LIN {X 0,Y 445.278,Z 563.704,A -85,B 0,C 180,E1 20681.751,E2 20681.751} C_VEL
LIN {X 0,Y 446.014,Z 547.85,A -85,B 0,C 180,E1 20680.554,E2 20680.554} C_VEL
LIN {X 0,Y 446.635,Z 530.926,A -85,B 0,C 180,E1 20679.559,E2 20679.559} C_VEL
LIN {X 0,Y 447.095,Z 513.78,A -85,B 0,C 180,E1 20678.817,E2 20678.817} C_VEL
LIN {X 0,Y 447.348,Z 495.46,A -85,B 0,C 180,E1 20678.284,E2 20678.284} C_VEL
LIN {X 0,Y 449.909,Z 332.781,A -85,B 0,C 180,E1 20675.326,E2 20675.326} C_VEL
LIN {X 0,Y 449.103,Z 327.513,A -85,B 0,C 180,E1 20675.165,E2 20675.165} C_VEL
LIN {X 0,Y 450.293,Z 289.121,A -85,B 0,C 180,E1 20671.484,E2 20671.484} C_VEL
LIN {X 0,Y 450.643,Z 279.918,A -85,B 0,C 180,E1 20670.582,E2 20670.582} C_VEL
LIN {X 0,Y 452.131,Z 281.25,A -85,B 0,C 180,E1 20670.354,E2 20670.354} C_VEL
LIN {X 0,Y 454.578,Z 280.888,A -85,B 0,C 180,E1 20670.046,E2 20670.046} C_VEL
LIN {X 0,Y 458.108,Z 278.184,A -85,B 0,C 180,E1 20669.668,E2 20669.668} C_VEL
LIN {X 0,Y 459.445,Z 277.014,A -85,B 0,C 180,E1 20669.531,E2 20669.531} C_VEL
LIN {X 0,Y 463.235,Z 276.31,A -85,B 0,C 180,E1 20669.089,E2 20669.089} C_VEL
LIN {X 0,Y 467.513,Z 273.586,A -85,B 0,C 180,E1 20668.652,E2 20668.652} C_VEL
LIN {X 0,Y 468.934,Z 272.801,A -85,B 0,C 180,E1 20668.507,E2 20668.507} C_VEL
LIN {X 0,Y 471.015,Z 272.513,A -85,B 0,C 180,E1 20668.278,E2 20668.278} C_VEL
LIN {X 0,Y 466.209,Z 421.313,A -85,B 0,C 180,E1 20665.555,E2 20665.555} C_VEL
LIN {X 0,Y 465.176,Z 428.993,A -85,B 0,C 180,E1 20665.49,E2 20665.49} C_VEL
LIN {X 0,Y 459.547,Z 449.472,A -85,B 0,C 180,E1 20665.582,E2 20665.582} C_VEL
LIN {X 0,Y 458.739,Z 456.06,A -85,B 0,C 180,E1 20665.515,E2 20665.515} C_VEL
LIN {X 0,Y 457.752,Z 483.582,A -85,B 0,C 180,E1 20664.917,E2 20664.917} C_VEL
LIN {X 0,Y 456.588,Z 504.2,A -85,B 0,C 180,E1 20664.247,E2 20664.247} C_VEL
LIN {X 0,Y 454.896,Z 524.708,A -85,B 0,C 180,E1 20663.348,E2 20663.348} C_VEL
LIN {X 0,Y 452.943,Z 544.086,A -85,B 0,C 180,E1 20662.268,E2 20662.268} C_VEL
LIN {X 0,Y 450.644,Z 563.469,A -85,B 0,C 180,E1 20660.94,E2 20660.94} C_VEL
LIN {X 0,Y 448.195,Z 581.756,A -85,B 0,C 180,E1 20659.43,E2 20659.43} C_VEL
LIN {X 0,Y 445.575,Z 599.353,A -85,B 0,C 180,E1 20657.685,E2 20657.685} C_VEL
LIN {X 0,Y 443.037,Z 615.611,A -85,B 0,C 180,E1 20655.784,E2 20655.784} C_VEL
LIN {X 0,Y 440.527,Z 631.382,A -85,B 0,C 180,E1 20653.611,E2 20653.611} C_VEL
LIN {X 0,Y 438.339,Z 645.243,A -85,B 0,C 180,E1 20651.369,E2 20651.369} C_VEL
LIN {X 0,Y 436.373,Z 658.158,A -85,B 0,C 180,E1 20648.89,E2 20648.89} C_VEL
LIN {X 0,Y 434.733,Z 670.08,A -85,B 0,C 180,E1 20646.168,E2 20646.168} C_VEL
LIN {X 0,Y 433.546,Z 679.999,A -85,B 0,C 180,E1 20643.449,E2 20643.449} C_VEL
LIN {X 0,Y 432.699,Z 688.525,A -85,B 0,C 180,E1 20640.555,E2 20640.555} C_VEL
LIN {X 0,Y 432.258,Z 694.523,A -85,B 0,C 180,E1 20638.006,E2 20638.006} C_VEL
LIN {X 0,Y 432.009,Z 700.325,A -85,B 0,C 180,E1 20634.869,E2 20634.869} C_VEL
LIN {X 0,Y 431.939,Z 703.61,A -85,B 0,C 180,E1 20632.311,E2 20632.311} C_VEL
LIN {X 0,Y 431.908,Z 705.568,A -85,B 0,C 180,E1 20629.896,E2 20629.896} C_VEL
LIN {X 0,Y 431.906,Z 706.457,A -85,B 0,C 180,E1 20627.237,E2 20627.237} C_VEL
LIN {X 0,Y 431.914,Z 705.763,A -85,B 0,C 180,E1 20624.342,E2 20624.342} C_VEL
LIN {X 0,Y 431.928,Z 703.903,A -85,B 0,C 180,E1 20621.89,E2 20621.89} C_VEL
LIN {X 0,Y 431.98,Z 700.918,A -85,B 0,C 180,E1 20619.459,E2 20619.459} C_VEL
LIN {X 0,Y 432.211,Z 695.519,A -85,B 0,C 180,E1 20616.376,E2 20616.376} C_VEL
LIN {X 0,Y 432.599,Z 689.749,A -85,B 0,C 180,E1 20613.843,E2 20613.843} C_VEL
LIN {X 0,Y 433.329,Z 681.908,A -85,B 0,C 180,E1 20611.058,E2 20611.058} C_VEL
LIN {X 0,Y 434.437,Z 672.167,A -85,B 0,C 180,E1 20608.286,E2 20608.286} C_VEL
LIN {X 0,Y 435.841,Z 661.693,A -85,B 0,C 180,E1 20605.79,E2 20605.79} C_VEL
LIN {X 0,Y 437.776,Z 648.664,A -85,B 0,C 180,E1 20603.179,E2 20603.179} C_VEL
LIN {X 0,Y 440.074,Z 634.053,A -85,B 0,C 180,E1 20600.717,E2 20600.717} C_VEL
LIN {X 0,Y 442.535,Z 618.775,A -85,B 0,C 180,E1 20598.532,E2 20598.532} C_VEL
LIN {X 0,Y 445.057,Z 602.818,A -85,B 0,C 180,E1 20596.601,E2 20596.601} C_VEL
LIN {X 0,Y 447.614,Z 585.784,A -85,B 0,C 180,E1 20594.85,E2 20594.85} C_VEL
LIN {X 0,Y 450.175,Z 567.801,A -85,B 0,C 180,E1 20593.284,E2 20593.284} C_VEL
LIN {X 0,Y 452.464,Z 549.874,A -85,B 0,C 180,E1 20591.979,E2 20591.979} C_VEL
LIN {X 0,Y 454.464,Z 531.263,A -85,B 0,C 180,E1 20590.864,E2 20590.864} C_VEL
LIN {X 0,Y 456.333,Z 510.862,A -85,B 0,C 180,E1 20589.879,E2 20589.879} C_VEL
LIN {X 0,Y 457.832,Z 489.947,A -85,B 0,C 180,E1 20589.109,E2 20589.109} C_VEL
LIN {X 0,Y 458.748,Z 469.432,A -85,B 0,C 180,E1 20588.58,E2 20588.58} C_VEL
LIN {X 0,Y 465.748,Z 266.596,A -85,B 0,C 180,E1 20584.795,E2 20584.795} C_VEL
LIN {X 0,Y 466.581,Z 237.059,A -85,B 0,C 180,E1 20584.241,E2 20584.241} C_VEL
LIN {X 0,Y 453.17,Z 217.007,A -85,B 0,C 180,E1 20582.222,E2 20582.222} C_VEL
LIN {X 0,Y 445.587,Z 207.661,A -85,B 0,C 180,E1 20581.061,E2 20581.061} C_VEL
LIN {X 0,Y 440.176,Z 201.25,A -85,B 0,C 180,E1 20580.168,E2 20580.168} C_VEL
LIN {X 0,Y 437.829,Z 196.904,A -85,B 0,C 180,E1 20579.168,E2 20579.168} C_VEL
LIN {X 0,Y 435.976,Z 193.053,A -85,B 0,C 180,E1 20578.305,E2 20578.305} C_VEL
LIN {X 0,Y 433.608,Z 189.423,A -85,B 0,C 180,E1 20577.345,E2 20577.345} C_VEL
LIN {X 0,Y 433.237,Z 187.766,A -85,B 0,C 180,E1 20576.999,E2 20576.999} C_VEL
LIN {X 0,Y 433.227,Z 187.768,A -85,B 0,C 180,E1 20573.126,E2 20573.126} C_VEL
LIN {X 0,Y 433.243,Z 187.762,A -85,B 0,C 180,E1 20569.397,E2 20569.397} C_VEL
LIN {X 0,Y 433.252,Z 187.758,A -85,B 0,C 180,E1 20565.632,E2 20565.632} C_VEL
LIN {X 0,Y 433.251,Z 187.759,A -85,B 0,C 180,E1 20561.805,E2 20561.805} C_VEL
LIN {X 0,Y 433.236,Z 187.766,A -85,B 0,C 180,E1 20558.04,E2 20558.04} C_VEL
LIN {X 0,Y 433.219,Z 187.773,A -85,B 0,C 180,E1 20554.274,E2 20554.274} C_VEL
LIN {X 0,Y 433.244,Z 187.764,A -85,B 0,C 180,E1 20550.513,E2 20550.513} C_VEL
LIN {X 0,Y 433.259,Z 187.752,A -85,B 0,C 180,E1 20546.734,E2 20546.734} C_VEL
LIN {X 0,Y 433.251,Z 187.746,A -85,B 0,C 180,E1 20542.955,E2 20542.955} C_VEL
LIN {X 0,Y 433.235,Z 187.76,A -85,B 0,C 180,E1 20539.131,E2 20539.131} C_VEL
LIN {X 0,Y 433.207,Z 187.773,A -85,B 0,C 180,E1 20535.393,E2 20535.393} C_VEL
LIN {X 0,Y 433.2,Z 187.772,A -85,B 0,C 180,E1 20531.584,E2 20531.584} C_VEL
LIN {X 0,Y 433.222,Z 187.759,A -85,B 0,C 180,E1 20527.827,E2 20527.827} C_VEL
LIN {X 0,Y 433.245,Z 187.748,A -85,B 0,C 180,E1 20524.103,E2 20524.103} C_VEL
LIN {X 0,Y 433.258,Z 187.751,A -85,B 0,C 180,E1 20520.265,E2 20520.265} C_VEL
LIN {X 0,Y 433.251,Z 187.755,A -85,B 0,C 180,E1 20516.428,E2 20516.428} C_VEL
LIN {X 0,Y 433.235,Z 187.757,A -85,B 0,C 180,E1 20512.575,E2 20512.575} C_VEL
LIN {X 0,Y 433.248,Z 187.755,A -85,B 0,C 180,E1 20508.761,E2 20508.761} C_VEL
LIN {X 0,Y 433.262,Z 187.753,A -85,B 0,C 180,E1 20505.021,E2 20505.021} C_VEL
LIN {X 0,Y 433.248,Z 187.756,A -85,B 0,C 180,E1 20501.15,E2 20501.15} C_VEL
LIN {X 0,Y 433.488,Z 188.953,A -85,B 0,C 180,E1 20500.882,E2 20500.882} C_VEL
LIN {X 0,Y 435.26,Z 192.141,A -85,B 0,C 180,E1 20500.125,E2 20500.125} C_VEL
LIN {X 0,Y 436.158,Z 193.757,A -85,B 0,C 180,E1 20499.748,E2 20499.748} C_VEL
LIN {X 0,Y 438.842,Z 198.769,A -85,B 0,C 180,E1 20498.621,E2 20498.621} C_VEL
LIN {X 0,Y 443.751,Z 208.113,A -85,B 0,C 180,E1 20496.637,E2 20496.637} C_VEL
LIN {X 0,Y 450.114,Z 220.548,A -85,B 0,C 180,E1 20494.191,E2 20494.191} C_VEL
LIN {X 0,Y 458.928,Z 239.006,A -85,B 0,C 180,E1 20490.932,E2 20490.932} C_VEL
LIN {X 0,Y 465.596,Z 254.171,A -85,B 0,C 180,E1 20488.522,E2 20488.522} C_VEL
LIN {X 0,Y 461.582,Z 295.714,A -85,B 0,C 180,E1 20484.966,E2 20484.966} C_VEL
LIN {X 0,Y 460.595,Z 316.537,A -85,B 0,C 180,E1 20483.114,E2 20483.114} C_VEL
LIN {X 0,Y 461.621,Z 333.917,A -85,B 0,C 180,E1 20481.406,E2 20481.406} C_VEL
LIN {X 0,Y 464.524,Z 349.654,A -85,B 0,C 180,E1 20479.699,E2 20479.699} C_VEL
LIN {X 0,Y 469.216,Z 363.952,A -85,B 0,C 180,E1 20478.002,E2 20478.002} C_VEL
LIN {X 0,Y 475.939,Z 377.183,A -85,B 0,C 180,E1 20476.276,E2 20476.276} C_VEL
LIN {X 0,Y 484.496,Z 388.72,A -85,B 0,C 180,E1 20474.604,E2 20474.604} C_VEL
LIN {X 0,Y 493.529,Z 397.655,A -85,B 0,C 180,E1 20473.17,E2 20473.17} C_VEL
LIN {X 0,Y 501.232,Z 403.797,A -85,B 0,C 180,E1 20472.107,E2 20472.107} C_VEL
LIN {X 0,Y 490.067,Z 420.572,A -85,B 0,C 180,E1 20471.613,E2 20471.613} C_VEL
LIN {X 0,Y 481.918,Z 435.231,A -85,B 0,C 180,E1 20471.045,E2 20471.045} C_VEL
LIN {X 0,Y 472.016,Z 452.159,A -85,B 0,C 180,E1 20470.405,E2 20470.405} C_VEL
LIN {X 0,Y 465.347,Z 466.548,A -85,B 0,C 180,E1 20469.718,E2 20469.718} C_VEL
LIN {X 0,Y 463.803,Z 470.28,A -85,B 0,C 180,E1 20469.564,E2 20469.564} C_VEL
LIN {X 0,Y 461.689,Z 487.127,A -85,B 0,C 180,E1 20469.443,E2 20469.443} C_VEL
LIN {X 0,Y 460.843,Z 502.83,A -85,B 0,C 180,E1 20469.212,E2 20469.212} C_VEL
LIN {X 0,Y 459.439,Z 528.442,A -85,B 0,C 180,E1 20468.647,E2 20468.647} C_VEL
LIN {X 0,Y 457.323,Z 552.538,A -85,B 0,C 180,E1 20467.905,E2 20467.905} C_VEL
LIN {X 0,Y 455.012,Z 575.297,A -85,B 0,C 180,E1 20466.962,E2 20466.962} C_VEL
LIN {X 0,Y 452.552,Z 597.1,A -85,B 0,C 180,E1 20465.822,E2 20465.822} C_VEL
LIN {X 0,Y 449.961,Z 618.518,A -85,B 0,C 180,E1 20464.446,E2 20464.446} C_VEL
LIN {X 0,Y 447.255,Z 639.445,A -85,B 0,C 180,E1 20462.828,E2 20462.828} C_VEL
LIN {X 0,Y 444.794,Z 657.926,A -85,B 0,C 180,E1 20461.132,E2 20461.132} C_VEL
LIN {X 0,Y 442.362,Z 675.786,A -85,B 0,C 180,E1 20459.223,E2 20459.223} C_VEL
LIN {X 0,Y 439.987,Z 693.254,A -85,B 0,C 180,E1 20457.026,E2 20457.026} C_VEL
LIN {X 0,Y 437.78,Z 709.815,A -85,B 0,C 180,E1 20454.562,E2 20454.562} C_VEL
LIN {X 0,Y 436.1,Z 723.144,A -85,B 0,C 180,E1 20452.228,E2 20452.228} C_VEL
LIN {X 0,Y 434.714,Z 735.279,A -85,B 0,C 180,E1 20449.761,E2 20449.761} C_VEL
LIN {X 0,Y 433.525,Z 747.008,A -85,B 0,C 180,E1 20446.894,E2 20446.894} C_VEL
LIN {X 0,Y 432.771,Z 756.133,A -85,B 0,C 180,E1 20444.176,E2 20444.176} C_VEL
LIN {X 0,Y 432.304,Z 763.48,A -85,B 0,C 180,E1 20441.473,E2 20441.473} C_VEL
LIN {X 0,Y 432.036,Z 769.389,A -85,B 0,C 180,E1 20438.517,E2 20438.517} C_VEL
LIN {X 0,Y 431.937,Z 773.513,A -85,B 0,C 180,E1 20435.516,E2 20435.516} C_VEL
LIN {X 0,Y 431.91,Z 775.786,A -85,B 0,C 180,E1 20432.654,E2 20432.654} C_VEL
LIN {X 0,Y 431.909,Z 776.489,A -85,B 0,C 180,E1 20429.867,E2 20429.867} C_VEL
LIN {X 0,Y 431.914,Z 775.58,A -85,B 0,C 180,E1 20426.948,E2 20426.948} C_VEL
LIN {X 0,Y 431.941,Z 773.135,A -85,B 0,C 180,E1 20424.154,E2 20424.154} C_VEL
LIN {X 0,Y 432.039,Z 769.149,A -85,B 0,C 180,E1 20421.348,E2 20421.348} C_VEL
LIN {X 0,Y 432.304,Z 763.48,A -85,B 0,C 180,E1 20418.527,E2 20418.527} C_VEL
LIN {X 0,Y 432.77,Z 756.108,A -85,B 0,C 180,E1 20415.824,E2 20415.824} C_VEL
LIN {X 0,Y 433.524,Z 746.91,A -85,B 0,C 180,E1 20413.106,E2 20413.106} C_VEL
LIN {X 0,Y 434.575,Z 736.284,A -85,B 0,C 180,E1 20410.512,E2 20410.512} C_VEL
LIN {X 0,Y 436,Z 723.467,A -85,B 0,C 180,E1 20407.891,E2 20407.891} C_VEL
LIN {X 0,Y 437.791,Z 708.789,A -85,B 0,C 180,E1 20405.364,E2 20405.364} C_VEL
LIN {X 0,Y 439.903,Z 692.262,A -85,B 0,C 180,E1 20402.962,E2 20402.962} C_VEL
LIN {X 0,Y 442.224,Z 674.463,A -85,B 0,C 180,E1 20400.766,E2 20400.766} C_VEL
LIN {X 0,Y 444.649,Z 655.737,A -85,B 0,C 180,E1 20398.812,E2 20398.812} C_VEL
LIN {X 0,Y 447.103,Z 636.244,A -85,B 0,C 180,E1 20397.083,E2 20397.083} C_VEL
LIN {X 0,Y 449.739,Z 614.493,A -85,B 0,C 180,E1 20395.464,E2 20395.464} C_VEL
LIN {X 0,Y 452.221,Z 593.005,A -85,B 0,C 180,E1 20394.132,E2 20394.132} C_VEL
LIN {X 0,Y 454.598,Z 570.635,A -85,B 0,C 180,E1 20393.011,E2 20393.011} C_VEL
LIN {X 0,Y 456.965,Z 546.335,A -85,B 0,C 180,E1 20392.049,E2 20392.049} C_VEL
LIN {X 0,Y 459.06,Z 521.772,A -85,B 0,C 180,E1 20391.33,E2 20391.33} C_VEL
LIN {X 0,Y 460.256,Z 496.354,A -85,B 0,C 180,E1 20390.796,E2 20390.796} C_VEL
LIN {X 0,Y 461.919,Z 471.592,A -85,B 0,C 180,E1 20390.479,E2 20390.479} C_VEL
LIN {X 0,Y 463.271,Z 461.084,A -85,B 0,C 180,E1 20390.374,E2 20390.374} C_VEL
LIN {X 0,Y 468.481,Z 442.909,A -85,B 0,C 180,E1 20389.708,E2 20389.708} C_VEL
LIN {X 0,Y 474.364,Z 426.367,A -85,B 0,C 180,E1 20389.2,E2 20389.2} C_VEL
LIN {X 0,Y 480.138,Z 408.39,A -85,B 0,C 180,E1 20388.61,E2 20388.61} C_VEL
LIN {X 0,Y 489.341,Z 385.58,A -85,B 0,C 180,E1 20388.027,E2 20388.027} C_VEL
LIN {X 0,Y 502.922,Z 356.818,A -85,B 0,C 180,E1 20387.471,E2 20387.471} C_VEL
LIN {X 0,Y 509.045,Z 344.473,A -85,B 0,C 180,E1 20387.263,E2 20387.263} C_VEL
LIN {X 0,Y 515.527,Z 326.752,A -85,B 0,C 180,E1 20386.792,E2 20386.792} C_VEL
LIN {X 0,Y 518.84,Z 318.413,A -85,B 0,C 180,E1 20386.595,E2 20386.595} C_VEL
LIN {X 0,Y 502.17,Z 306.197,A -85,B 0,C 180,E1 20384.495,E2 20384.495} C_VEL
LIN {X 0,Y 493.129,Z 297.375,A -85,B 0,C 180,E1 20383.101,E2 20383.101} C_VEL
LIN {X 0,Y 484.783,Z 286.271,A -85,B 0,C 180,E1 20381.523,E2 20381.523} C_VEL
LIN {X 0,Y 478.266,Z 273.614,A -85,B 0,C 180,E1 20379.927,E2 20379.927} C_VEL
LIN {X 0,Y 469.301,Z 252.138,A -85,B 0,C 180,E1 20377.233,E2 20377.233} C_VEL
LIN {X 0,Y 462.525,Z 238.077,A -85,B 0,C 180,E1 20375.158,E2 20375.158} C_VEL
LIN {X 0,Y 458.445,Z 240.134,A -85,B 0,C 180,E1 20374.696,E2 20374.696} C_VEL
LIN {X 0,Y 454.514,Z 242.602,A -85,B 0,C 180,E1 20374.274,E2 20374.274} C_VEL
LIN {X 0,Y 452.137,Z 243.649,A -85,B 0,C 180,E1 20373.975,E2 20373.975} C_VEL
LIN {X 0,Y 449.086,Z 245.963,A -85,B 0,C 180,E1 20373.668,E2 20373.668} C_VEL
LIN {X 0,Y 446.403,Z 246.739,A -85,B 0,C 180,E1 20373.281,E2 20373.281} C_VEL
LIN {X 0,Y 446.039,Z 246.86,A -85,B 0,C 180,E1 20373.197,E2 20373.197} C_VEL
LIN {X 0,Y 445.836,Z 284.892,A -85,B 0,C 180,E1 20370.007,E2 20370.007} C_VEL
LIN {X 0,Y 445.36,Z 320.307,A -85,B 0,C 180,E1 20366.964,E2 20366.964} C_VEL
LIN {X 0,Y 444.853,Z 337.961,A -85,B 0,C 180,E1 20365.422,E2 20365.422} C_VEL
LIN {X 0,Y 443.334,Z 344.859,A -85,B 0,C 180,E1 20364.98,E2 20364.98} C_VEL
LIN {X 0,Y 440.387,Z 449.833,A -85,B 0,C 180,E1 20362.799,E2 20362.799} C_VEL
LIN {X 0,Y 439.712,Z 505.996,A -85,B 0,C 180,E1 20361.711,E2 20361.711} C_VEL
LIN {X 0,Y 439.647,Z 524.324,A -85,B 0,C 180,E1 20361.151,E2 20361.151} C_VEL
LIN {X 0,Y 439.386,Z 540.119,A -85,B 0,C 180,E1 20360.444,E2 20360.444} C_VEL
LIN {X 0,Y 438.913,Z 555.89,A -85,B 0,C 180,E1 20359.495,E2 20359.495} C_VEL
LIN {X 0,Y 438.303,Z 570.746,A -85,B 0,C 180,E1 20358.349,E2 20358.349} C_VEL
LIN {X 0,Y 437.584,Z 584.595,A -85,B 0,C 180,E1 20357.006,E2 20357.006} C_VEL
LIN {X 0,Y 436.81,Z 597.133,A -85,B 0,C 180,E1 20355.49,E2 20355.49} C_VEL
LIN {X 0,Y 436.025,Z 608.481,A -85,B 0,C 180,E1 20353.797,E2 20353.797} C_VEL
LIN {X 0,Y 435.34,Z 617.843,A -85,B 0,C 180,E1 20352.063,E2 20352.063} C_VEL
LIN {X 0,Y 434.701,Z 626.354,A -85,B 0,C 180,E1 20350.067,E2 20350.067} C_VEL
LIN {X 0,Y 434.178,Z 633.269,A -85,B 0,C 180,E1 20347.942,E2 20347.942} C_VEL
LIN {X 0,Y 433.796,Z 638.259,A -85,B 0,C 180,E1 20345.82,E2 20345.82} C_VEL
LIN {X 0,Y 433.52,Z 641.592,A -85,B 0,C 180,E1 20343.57,E2 20343.57} C_VEL
LIN {X 0,Y 433.359,Z 643.129,A -85,B 0,C 180,E1 20341.322,E2 20341.322} C_VEL
LIN {X 0,Y 433.283,Z 642.929,A -85,B 0,C 180,E1 20339.074,E2 20339.074} C_VEL
LIN {X 0,Y 433.283,Z 640.94,A -85,B 0,C 180,E1 20336.825,E2 20336.825} C_VEL
LIN {X 0,Y 433.384,Z 637.159,A -85,B 0,C 180,E1 20334.572,E2 20334.572} C_VEL
LIN {X 0,Y 433.627,Z 631.501,A -85,B 0,C 180,E1 20332.314,E2 20332.314} C_VEL
LIN {X 0,Y 434,Z 624.186,A -85,B 0,C 180,E1 20330.184,E2 20330.184} C_VEL
LIN {X 0,Y 434.503,Z 615.365,A -85,B 0,C 180,E1 20328.182,E2 20328.182} C_VEL
LIN {X 0,Y 435.149,Z 605.088,A -85,B 0,C 180,E1 20326.31,E2 20326.31} C_VEL
LIN {X 0,Y 435.903,Z 593.254,A -85,B 0,C 180,E1 20324.569,E2 20324.569} C_VEL
LIN {X 0,Y 436.728,Z 579.803,A -85,B 0,C 180,E1 20322.959,E2 20322.959} C_VEL
LIN {X 0,Y 437.561,Z 565.232,A -85,B 0,C 180,E1 20321.542,E2 20321.542} C_VEL
LIN {X 0,Y 438.318,Z 549.639,A -85,B 0,C 180,E1 20320.338,E2 20320.338} C_VEL
LIN {X 0,Y 438.965,Z 532.854,A -85,B 0,C 180,E1 20319.325,E2 20319.325} C_VEL
LIN {X 0,Y 439.457,Z 515.59,A -85,B 0,C 180,E1 20318.551,E2 20318.551} C_VEL
LIN {X 0,Y 439.727,Z 497.468,A -85,B 0,C 180,E1 20318.004,E2 20318.004} C_VEL
LIN {X 0,Y 442.496,Z 333.853,A -85,B 0,C 180,E1 20314.953,E2 20314.953} C_VEL
LIN {X 0,Y 441.682,Z 328.347,A -85,B 0,C 180,E1 20314.776,E2 20314.776} C_VEL
LIN {X 0,Y 442.901,Z 292.617,A -85,B 0,C 180,E1 20311.314,E2 20311.314} C_VEL
LIN {X 0,Y 444.403,Z 293.909,A -85,B 0,C 180,E1 20311.07,E2 20311.07} C_VEL
LIN {X 0,Y 446.798,Z 293.524,A -85,B 0,C 180,E1 20310.756,E2 20310.756} C_VEL
LIN {X 0,Y 450.335,Z 290.682,A -85,B 0,C 180,E1 20310.359,E2 20310.359} C_VEL
LIN {X 0,Y 451.768,Z 289.242,A -85,B 0,C 180,E1 20310.207,E2 20310.207} C_VEL
LIN {X 0,Y 455.5,Z 288.479,A -85,B 0,C 180,E1 20309.75,E2 20309.75} C_VEL
LIN {X 0,Y 459.711,Z 285.708,A -85,B 0,C 180,E1 20309.297,E2 20309.297} C_VEL
LIN {X 0,Y 460.74,Z 284.85,A -85,B 0,C 180,E1 20309.193,E2 20309.193} C_VEL
LIN {X 0,Y 464.761,Z 283.865,A -85,B 0,C 180,E1 20308.739,E2 20308.739} C_VEL
LIN {X 0,Y 458.739,Z 456.06,A -85,B 0,C 180,E1 20305.515,E2 20305.515} C_VEL
LIN {X 0,Y 457.686,Z 463.731,A -85,B 0,C 180,E1 20305.445,E2 20305.445} C_VEL
LIN {X 0,Y 452.108,Z 483.056,A -85,B 0,C 180,E1 20305.476,E2 20305.476} C_VEL
LIN {X 0,Y 450.994,Z 490.635,A -85,B 0,C 180,E1 20305.325,E2 20305.325} C_VEL
LIN {X 0,Y 449.552,Z 511.65,A -85,B 0,C 180,E1 20304.561,E2 20304.561} C_VEL
LIN {X 0,Y 447.637,Z 532.684,A -85,B 0,C 180,E1 20303.547,E2 20303.547} C_VEL
LIN {X 0,Y 445.508,Z 551.937,A -85,B 0,C 180,E1 20302.377,E2 20302.377} C_VEL
LIN {X 0,Y 442.934,Z 571.13,A -85,B 0,C 180,E1 20300.944,E2 20300.944} C_VEL
LIN {X 0,Y 440.278,Z 589.146,A -85,B 0,C 180,E1 20299.324,E2 20299.324} C_VEL
LIN {X 0,Y 437.407,Z 607.125,A -85,B 0,C 180,E1 20297.397,E2 20297.397} C_VEL
LIN {X 0,Y 434.767,Z 623.041,A -85,B 0,C 180,E1 20295.38,E2 20295.38} C_VEL
LIN {X 0,Y 432.192,Z 638.327,A -85,B 0,C 180,E1 20293.094,E2 20293.094} C_VEL
LIN {X 0,Y 429.888,Z 652.138,A -85,B 0,C 180,E1 20290.636,E2 20290.636} C_VEL
LIN {X 0,Y 427.965,Z 664.336,A -85,B 0,C 180,E1 20288.062,E2 20288.062} C_VEL
LIN {X 0,Y 426.442,Z 675.281,A -85,B 0,C 180,E1 20285.319,E2 20285.319} C_VEL
LIN {X 0,Y 425.346,Z 684.309,A -85,B 0,C 180,E1 20282.569,E2 20282.569} C_VEL
LIN {X 0,Y 424.62,Z 691.72,A -85,B 0,C 180,E1 20279.792,E2 20279.792} C_VEL
LIN {X 0,Y 424.18,Z 698.095,A -85,B 0,C 180,E1 20276.7,E2 20276.7} C_VEL
LIN {X 0,Y 424.002,Z 702.077,A -85,B 0,C 180,E1 20274.077,E2 20274.077} C_VEL
LIN {X 0,Y 423.928,Z 705.101,A -85,B 0,C 180,E1 20271.153,E2 20271.153} C_VEL
LIN {X 0,Y 423.906,Z 706.436,A -85,B 0,C 180,E1 20268.283,E2 20268.283} C_VEL
LIN {X 0,Y 423.911,Z 706.462,A -85,B 0,C 180,E1 20265.774,E2 20265.774} C_VEL
LIN {X 0,Y 423.921,Z 705.235,A -85,B 0,C 180,E1 20262.948,E2 20262.948} C_VEL
LIN {X 0,Y 423.986,Z 702.35,A -85,B 0,C 180,E1 20260.05,E2 20260.05} C_VEL
LIN {X 0,Y 424.151,Z 698.485,A -85,B 0,C 180,E1 20257.45,E2 20257.45} C_VEL
LIN {X 0,Y 424.524,Z 692.839,A -85,B 0,C 180,E1 20254.593,E2 20254.593} C_VEL
LIN {X 0,Y 425.21,Z 685.453,A -85,B 0,C 180,E1 20251.752,E2 20251.752} C_VEL
LIN {X 0,Y 426.263,Z 676.395,A -85,B 0,C 180,E1 20248.925,E2 20248.925} C_VEL
LIN {X 0,Y 427.783,Z 665.412,A -85,B 0,C 180,E1 20246.114,E2 20246.114} C_VEL
LIN {X 0,Y 429.612,Z 653.691,A -85,B 0,C 180,E1 20243.586,E2 20243.586} C_VEL
LIN {X 0,Y 431.76,Z 640.548,A -85,B 0,C 180,E1 20241.209,E2 20241.209} C_VEL
LIN {X 0,Y 434.199,Z 626.151,A -85,B 0,C 180,E1 20238.981,E2 20238.981} C_VEL
LIN {X 0,Y 436.781,Z 611.003,A -85,B 0,C 180,E1 20236.969,E2 20236.969} C_VEL
LIN {X 0,Y 439.6,Z 593.786,A -85,B 0,C 180,E1 20235.04,E2 20235.04} C_VEL
LIN {X 0,Y 442.263,Z 576.182,A -85,B 0,C 180,E1 20233.382,E2 20233.382} C_VEL
LIN {X 0,Y 444.921,Z 556.962,A -85,B 0,C 180,E1 20231.866,E2 20231.866} C_VEL
LIN {X 0,Y 447.286,Z 537.71,A -85,B 0,C 180,E1 20230.613,E2 20230.613} C_VEL
LIN {X 0,Y 449.205,Z 518.55,A -85,B 0,C 180,E1 20229.614,E2 20229.614} C_VEL
LIN {X 0,Y 450.848,Z 497.452,A -85,B 0,C 180,E1 20228.757,E2 20228.757} C_VEL
LIN {X 0,Y 452.03,Z 476.274,A -85,B 0,C 180,E1 20228.13,E2 20228.13} C_VEL
LIN {X 0,Y 459.235,Z 282.71,A -85,B 0,C 180,E1 20224.424,E2 20224.424} C_VEL
LIN {X 0,Y 460.607,Z 240.519,A -85,B 0,C 180,E1 20223.635,E2 20223.635} C_VEL
LIN {X 0,Y 446.908,Z 220.274,A -85,B 0,C 180,E1 20221.52,E2 20221.52} C_VEL
LIN {X 0,Y 435.31,Z 206.781,A -85,B 0,C 180,E1 20219.692,E2 20219.692} C_VEL
LIN {X 0,Y 433.557,Z 204.38,A -85,B 0,C 180,E1 20219.341,E2 20219.341} C_VEL
LIN {X 0,Y 430.863,Z 199.288,A -85,B 0,C 180,E1 20218.141,E2 20218.141} C_VEL
LIN {X 0,Y 428.345,Z 195.032,A -85,B 0,C 180,E1 20217.052,E2 20217.052} C_VEL
LIN {X 0,Y 427.57,Z 193.405,A -85,B 0,C 180,E1 20216.665,E2 20216.665} C_VEL
LIN {X 0,Y 425.579,Z 190.197,A -85,B 0,C 180,E1 20215.792,E2 20215.792} C_VEL
LIN {X 0,Y 425.264,Z 188.748,A -85,B 0,C 180,E1 20215.485,E2 20215.485} C_VEL
LIN {X 0,Y 425.272,Z 188.745,A -85,B 0,C 180,E1 20211.634,E2 20211.634} C_VEL
LIN {X 0,Y 425.292,Z 188.743,A -85,B 0,C 180,E1 20207.931,E2 20207.931} C_VEL
LIN {X 0,Y 425.31,Z 188.739,A -85,B 0,C 180,E1 20204.097,E2 20204.097} C_VEL
LIN {X 0,Y 425.322,Z 188.736,A -85,B 0,C 180,E1 20200.277,E2 20200.277} C_VEL
LIN {X 0,Y 425.308,Z 188.738,A -85,B 0,C 180,E1 20196.485,E2 20196.485} C_VEL
LIN {X 0,Y 425.298,Z 188.739,A -85,B 0,C 180,E1 20192.573,E2 20192.573} C_VEL
LIN {X 0,Y 425.326,Z 188.747,A -85,B 0,C 180,E1 20188.735,E2 20188.735} C_VEL
LIN {X 0,Y 425.32,Z 188.755,A -85,B 0,C 180,E1 20184.848,E2 20184.848} C_VEL
LIN {X 0,Y 425.306,Z 188.757,A -85,B 0,C 180,E1 20181.043,E2 20181.043} C_VEL
LIN {X 0,Y 425.281,Z 188.746,A -85,B 0,C 180,E1 20177.232,E2 20177.232} C_VEL
LIN {X 0,Y 425.254,Z 188.742,A -85,B 0,C 180,E1 20173.461,E2 20173.461} C_VEL
LIN {X 0,Y 425.274,Z 188.748,A -85,B 0,C 180,E1 20169.61,E2 20169.61} C_VEL
LIN {X 0,Y 425.299,Z 188.756,A -85,B 0,C 180,E1 20165.802,E2 20165.802} C_VEL
LIN {X 0,Y 425.316,Z 188.758,A -85,B 0,C 180,E1 20161.887,E2 20161.887} C_VEL
LIN {X 0,Y 425.319,Z 188.755,A -85,B 0,C 180,E1 20158.114,E2 20158.114} C_VEL
LIN {X 0,Y 425.298,Z 188.756,A -85,B 0,C 180,E1 20154.198,E2 20154.198} C_VEL
LIN {X 0,Y 425.304,Z 188.755,A -85,B 0,C 180,E1 20150.392,E2 20150.392} C_VEL
LIN {X 0,Y 425.324,Z 188.758,A -85,B 0,C 180,E1 20146.543,E2 20146.543} C_VEL
LIN {X 0,Y 425.318,Z 188.75,A -85,B 0,C 180,E1 20142.629,E2 20142.629} C_VEL
LIN {X 0,Y 425.545,Z 189.885,A -85,B 0,C 180,E1 20142.357,E2 20142.357} C_VEL
LIN {X 0,Y 427.225,Z 193.01,A -85,B 0,C 180,E1 20141.582,E2 20141.582} C_VEL
LIN {X 0,Y 428.166,Z 194.423,A -85,B 0,C 180,E1 20141.201,E2 20141.201} C_VEL
LIN {X 0,Y 430.179,Z 198.187,A -85,B 0,C 180,E1 20140.305,E2 20140.305} C_VEL
LIN {X 0,Y 433.996,Z 205.471,A -85,B 0,C 180,E1 20138.654,E2 20138.654} C_VEL
LIN {X 0,Y 440.2,Z 217.169,A -85,B 0,C 180,E1 20136.153,E2 20136.153} C_VEL
LIN {X 0,Y 448.127,Z 233.359,A -85,B 0,C 180,E1 20133.068,E2 20133.068} C_VEL
LIN {X 0,Y 456.787,Z 252.332,A -85,B 0,C 180,E1 20129.838,E2 20129.838} C_VEL
LIN {X 0,Y 459.212,Z 258.127,A -85,B 0,C 180,E1 20128.934,E2 20128.934} C_VEL
LIN {X 0,Y 454.082,Z 314.796,A -85,B 0,C 180,E1 20123.991,E2 20123.991} C_VEL
LIN {X 0,Y 454.576,Z 332.958,A -85,B 0,C 180,E1 20122.225,E2 20122.225} C_VEL
LIN {X 0,Y 456.874,Z 348.861,A -85,B 0,C 180,E1 20120.525,E2 20120.525} C_VEL
LIN {X 0,Y 461.078,Z 363.954,A -85,B 0,C 180,E1 20118.759,E2 20118.759} C_VEL
LIN {X 0,Y 466.877,Z 377.102,A -85,B 0,C 180,E1 20117.077,E2 20117.077} C_VEL
LIN {X 0,Y 473.845,Z 388.182,A -85,B 0,C 180,E1 20115.529,E2 20115.529} C_VEL
LIN {X 0,Y 483.549,Z 399.394,A -85,B 0,C 180,E1 20113.81,E2 20113.81} C_VEL
LIN {X 0,Y 491.877,Z 406.803,A -85,B 0,C 180,E1 20112.568,E2 20112.568} C_VEL
LIN {X 0,Y 481.462,Z 423.155,A -85,B 0,C 180,E1 20112.047,E2 20112.047} C_VEL
LIN {X 0,Y 474.216,Z 436.158,A -85,B 0,C 180,E1 20111.54,E2 20111.54} C_VEL
LIN {X 0,Y 465.308,Z 451.511,A -85,B 0,C 180,E1 20110.949,E2 20110.949} C_VEL
LIN {X 0,Y 458.076,Z 467.36,A -85,B 0,C 180,E1 20110.202,E2 20110.202} C_VEL
LIN {X 0,Y 455.772,Z 483.87,A -85,B 0,C 180,E1 20110.104,E2 20110.104} C_VEL
LIN {X 0,Y 454.677,Z 499.611,A -85,B 0,C 180,E1 20109.896,E2 20109.896} C_VEL
LIN {X 0,Y 453.243,Z 525.603,A -85,B 0,C 180,E1 20109.323,E2 20109.323} C_VEL
LIN {X 0,Y 450.989,Z 550.098,A -85,B 0,C 180,E1 20108.577,E2 20108.577} C_VEL
LIN {X 0,Y 448.503,Z 573.472,A -85,B 0,C 180,E1 20107.609,E2 20107.609} C_VEL
LIN {X 0,Y 445.884,Z 595.397,A -85,B 0,C 180,E1 20106.458,E2 20106.458} C_VEL
LIN {X 0,Y 443.101,Z 617.23,A -85,B 0,C 180,E1 20105.049,E2 20105.049} C_VEL
LIN {X 0,Y 440.367,Z 637.424,A -85,B 0,C 180,E1 20103.486,E2 20103.486} C_VEL
LIN {X 0,Y 437.64,Z 656.834,A -85,B 0,C 180,E1 20101.7,E2 20101.7} C_VEL
LIN {X 0,Y 435.145,Z 674.129,A -85,B 0,C 180,E1 20099.832,E2 20099.832} C_VEL
LIN {X 0,Y 432.621,Z 691.623,A -85,B 0,C 180,E1 20097.62,E2 20097.62} C_VEL
LIN {X 0,Y 430.293,Z 708.035,A -85,B 0,C 180,E1 20095.165,E2 20095.165} C_VEL
LIN {X 0,Y 428.469,Z 721.556,A -85,B 0,C 180,E1 20092.791,E2 20092.791} C_VEL
LIN {X 0,Y 426.901,Z 734.469,A -85,B 0,C 180,E1 20090.138,E2 20090.138} C_VEL
LIN {X 0,Y 425.627,Z 746.268,A -85,B 0,C 180,E1 20087.217,E2 20087.217} C_VEL
LIN {X 0,Y 424.797,Z 755.82,A -85,B 0,C 180,E1 20084.308,E2 20084.308} C_VEL
LIN {X 0,Y 424.317,Z 763.11,A -85,B 0,C 180,E1 20081.554,E2 20081.554} C_VEL
LIN {X 0,Y 424.042,Z 768.993,A -85,B 0,C 180,E1 20078.679,E2 20078.679} C_VEL
LIN {X 0,Y 423.939,Z 773.266,A -85,B 0,C 180,E1 20075.685,E2 20075.685} C_VEL
LIN {X 0,Y 423.914,Z 775.594,A -85,B 0,C 180,E1 20072.974,E2 20072.974} C_VEL
LIN {X 0,Y 423.913,Z 776.476,A -85,B 0,C 180,E1 20070,E2 20070} C_VEL
LIN {X 0,Y 423.914,Z 775.595,A -85,B 0,C 180,E1 20067.025,E2 20067.025} C_VEL
LIN {X 0,Y 423.939,Z 773.262,A -85,B 0,C 180,E1 20064.315,E2 20064.315} C_VEL
LIN {X 0,Y 424.038,Z 769.204,A -85,B 0,C 180,E1 20061.457,E2 20061.457} C_VEL
LIN {X 0,Y 424.298,Z 763.385,A -85,B 0,C 180,E1 20058.583,E2 20058.583} C_VEL
LIN {X 0,Y 424.767,Z 756.139,A -85,B 0,C 180,E1 20055.829,E2 20055.829} C_VEL
LIN {X 0,Y 425.555,Z 746.809,A -85,B 0,C 180,E1 20052.991,E2 20052.991} C_VEL
LIN {X 0,Y 426.677,Z 735.951,A -85,B 0,C 180,E1 20050.278,E2 20050.278} C_VEL
LIN {X 0,Y 428.162,Z 723.248,A -85,B 0,C 180,E1 20047.626,E2 20047.626} C_VEL
LIN {X 0,Y 430.109,Z 708.094,A -85,B 0,C 180,E1 20044.97,E2 20044.97} C_VEL
LIN {X 0,Y 432.278,Z 692.059,A -85,B 0,C 180,E1 20042.594,E2 20042.594} C_VEL
LIN {X 0,Y 434.672,Z 674.616,A -85,B 0,C 180,E1 20040.4,E2 20040.4} C_VEL
LIN {X 0,Y 437.217,Z 656.137,A -85,B 0,C 180,E1 20038.419,E2 20038.419} C_VEL
LIN {X 0,Y 439.739,Z 637.078,A -85,B 0,C 180,E1 20036.694,E2 20036.694} C_VEL
LIN {X 0,Y 442.509,Z 615.803,A -85,B 0,C 180,E1 20035.055,E2 20035.055} C_VEL
LIN {X 0,Y 445.088,Z 594.693,A -85,B 0,C 180,E1 20033.705,E2 20033.705} C_VEL
LIN {X 0,Y 447.792,Z 571.202,A -85,B 0,C 180,E1 20032.481,E2 20032.481} C_VEL
LIN {X 0,Y 450.255,Z 547.958,A -85,B 0,C 180,E1 20031.52,E2 20031.52} C_VEL
LIN {X 0,Y 452.512,Z 523.483,A -85,B 0,C 180,E1 20030.771,E2 20030.771} C_VEL
LIN {X 0,Y 454.037,Z 496.747,A -85,B 0,C 180,E1 20030.167,E2 20030.167} C_VEL
LIN {X 0,Y 455.703,Z 472.345,A -85,B 0,C 180,E1 20029.844,E2 20029.844} C_VEL
LIN {X 0,Y 457.302,Z 457.94,A -85,B 0,C 180,E1 20029.711,E2 20029.711} C_VEL
LIN {X 0,Y 462.975,Z 439.256,A -85,B 0,C 180,E1 20029.046,E2 20029.046} C_VEL
LIN {X 0,Y 468.058,Z 425.057,A -85,B 0,C 180,E1 20028.612,E2 20028.612} C_VEL
LIN {X 0,Y 474.355,Z 405.909,A -85,B 0,C 180,E1 20027.991,E2 20027.991} C_VEL
LIN {X 0,Y 483.878,Z 382.641,A -85,B 0,C 180,E1 20027.411,E2 20027.411} C_VEL
LIN {X 0,Y 497.912,Z 353.147,A -85,B 0,C 180,E1 20026.861,E2 20026.861} C_VEL
LIN {X 0,Y 502.938,Z 343,A -85,B 0,C 180,E1 20026.695,E2 20026.695} C_VEL
LIN {X 0,Y 509.964,Z 324.125,A -85,B 0,C 180,E1 20026.202,E2 20026.202} C_VEL
LIN {X 0,Y 510.447,Z 322.479,A -85,B 0,C 180,E1 20026.149,E2 20026.149} C_VEL
LIN {X 0,Y 494.704,Z 310.257,A -85,B 0,C 180,E1 20024.048,E2 20024.048} C_VEL
LIN {X 0,Y 485.171,Z 300.009,A -85,B 0,C 180,E1 20022.457,E2 20022.457} C_VEL
LIN {X 0,Y 477.749,Z 289.063,A -85,B 0,C 180,E1 20020.924,E2 20020.924} C_VEL
LIN {X 0,Y 470.539,Z 273.551,A -85,B 0,C 180,E1 20018.974,E2 20018.974} C_VEL
LIN {X 0,Y 463.362,Z 256.073,A -85,B 0,C 180,E1 20016.706,E2 20016.706} C_VEL
LIN {X 0,Y 458.75,Z 246.67,A -85,B 0,C 180,E1 20015.28,E2 20015.28} C_VEL
LIN {X 0,Y 454.01,Z 249.519,A -85,B 0,C 180,E1 20014.777,E2 20014.777} C_VEL
LIN {X 0,Y 452.572,Z 250.094,A -85,B 0,C 180,E1 20014.596,E2 20014.596} C_VEL
LIN {X 0,Y 448.536,Z 252.879,A -85,B 0,C 180,E1 20014.176,E2 20014.176} C_VEL
LIN {X 0,Y 445.619,Z 254.252,A -85,B 0,C 180,E1 20013.81,E2 20013.81} C_VEL
LIN {X 0,Y 442.246,Z 256.782,A -85,B 0,C 180,E1 20013.461,E2 20013.461} C_VEL
LIN {X 0,Y 439.69,Z 257.44,A -85,B 0,C 180,E1 20013.076,E2 20013.076} C_VEL
LIN {X 0,Y 439.494,Z 257.685,A -85,B 0,C 180,E1 20013.015,E2 20013.015} C_VEL
LIN {X 0,Y 439.02,Z 297.474,A -85,B 0,C 180,E1 20009.617,E2 20009.617} C_VEL
LIN {X 0,Y 438.219,Z 337.188,A -85,B 0,C 180,E1 20006.126,E2 20006.126} C_VEL
LIN {X 0,Y 437.769,Z 340.574,A -85,B 0,C 180,E1 20005.864,E2 20005.864} C_VEL
LIN {X 0,Y 436.306,Z 347.246,A -85,B 0,C 180,E1 20005.447,E2 20005.447} C_VEL
LIN {X 0,Y 433.07,Z 451.158,A -85,B 0,C 180,E1 20003.208,E2 20003.208} C_VEL
LIN {X 0,Y 432.287,Z 506.608,A -85,B 0,C 180,E1 20002.095,E2 20002.095} C_VEL
LIN {X 0,Y 432.224,Z 525.254,A -85,B 0,C 180,E1 20001.524,E2 20001.524} C_VEL
LIN {X 0,Y 431.957,Z 541.108,A -85,B 0,C 180,E1 20000.812,E2 20000.812} C_VEL
LIN {X 0,Y 431.453,Z 557.001,A -85,B 0,C 180,E1 19999.846,E2 19999.846} C_VEL
LIN {X 0,Y 430.774,Z 572.78,A -85,B 0,C 180,E1 19998.611,E2 19998.611} C_VEL
LIN {X 0,Y 430.01,Z 586.554,A -85,B 0,C 180,E1 19997.245,E2 19997.245} C_VEL
LIN {X 0,Y 429.172,Z 599.198,A -85,B 0,C 180,E1 19995.679,E2 19995.679} C_VEL
LIN {X 0,Y 428.325,Z 610.734,A -85,B 0,C 180,E1 19993.912,E2 19993.912} C_VEL
LIN {X 0,Y 427.598,Z 619.961,A -85,B 0,C 180,E1 19992.148,E2 19992.148} C_VEL
LIN {X 0,Y 426.915,Z 628.324,A -85,B 0,C 180,E1 19990.116,E2 19990.116} C_VEL
LIN {X 0,Y 426.357,Z 635.115,A -85,B 0,C 180,E1 19987.953,E2 19987.953} C_VEL
LIN {X 0,Y 425.946,Z 639.967,A -85,B 0,C 180,E1 19985.793,E2 19985.793} C_VEL
LIN {X 0,Y 425.65,Z 643.169,A -85,B 0,C 180,E1 19983.501,E2 19983.501} C_VEL
LIN {X 0,Y 425.478,Z 644.573,A -85,B 0,C 180,E1 19981.211,E2 19981.211} C_VEL
LIN {X 0,Y 425.395,Z 644.201,A -85,B 0,C 180,E1 19978.922,E2 19978.922} C_VEL
LIN {X 0,Y 425.397,Z 642.023,A -85,B 0,C 180,E1 19976.631,E2 19976.631} C_VEL
LIN {X 0,Y 425.515,Z 638.072,A -85,B 0,C 180,E1 19974.336,E2 19974.336} C_VEL
LIN {X 0,Y 425.762,Z 632.601,A -85,B 0,C 180,E1 19972.171,E2 19972.171} C_VEL
LIN {X 0,Y 426.159,Z 625.165,A -85,B 0,C 180,E1 19970.001,E2 19970.001} C_VEL
LIN {X 0,Y 426.697,Z 616.229,A -85,B 0,C 180,E1 19967.962,E2 19967.962} C_VEL
LIN {X 0,Y 427.383,Z 605.818,A -85,B 0,C 180,E1 19966.056,E2 19966.056} C_VEL
LIN {X 0,Y 428.177,Z 593.798,A -85,B 0,C 180,E1 19964.283,E2 19964.283} C_VEL
LIN {X 0,Y 429.05,Z 580.17,A -85,B 0,C 180,E1 19962.644,E2 19962.644} C_VEL
LIN {X 0,Y 429.877,Z 566.2,A -85,B 0,C 180,E1 19961.277,E2 19961.277} C_VEL
LIN {X 0,Y 430.671,Z 550.404,A -85,B 0,C 180,E1 19960.045,E2 19960.045} C_VEL
LIN {X 0,Y 431.349,Z 533.497,A -85,B 0,C 180,E1 19959.014,E2 19959.014} C_VEL
LIN {X 0,Y 431.854,Z 516.157,A -85,B 0,C 180,E1 19958.232,E2 19958.232} C_VEL
LIN {X 0,Y 432.137,Z 497.723,A -85,B 0,C 180,E1 19957.673,E2 19957.673} C_VEL
LIN {X 0,Y 435.093,Z 334.97,A -85,B 0,C 180,E1 19954.573,E2 19954.573} C_VEL
LIN {X 0,Y 434.276,Z 329.471,A -85,B 0,C 180,E1 19954.401,E2 19954.401} C_VEL
LIN {X 0,Y 435.196,Z 305.787,A -85,B 0,C 180,E1 19952.069,E2 19952.069} C_VEL
LIN {X 0,Y 436.748,Z 306.973,A -85,B 0,C 180,E1 19951.811,E2 19951.811} C_VEL
LIN {X 0,Y 439.334,Z 306.253,A -85,B 0,C 180,E1 19951.46,E2 19951.46} C_VEL
LIN {X 0,Y 443.04,Z 302.882,A -85,B 0,C 180,E1 19951.028,E2 19951.028} C_VEL
LIN {X 0,Y 444.129,Z 301.907,A -85,B 0,C 180,E1 19950.903,E2 19950.903} C_VEL
LIN {X 0,Y 447.815,Z 301.046,A -85,B 0,C 180,E1 19950.433,E2 19950.433} C_VEL
LIN {X 0,Y 452.165,Z 297.949,A -85,B 0,C 180,E1 19949.943,E2 19949.943} C_VEL
LIN {X 0,Y 453.531,Z 296.955,A -85,B 0,C 180,E1 19949.793,E2 19949.793} C_VEL
LIN {X 0,Y 458.508,Z 295.036,A -85,B 0,C 180,E1 19949.226,E2 19949.226} C_VEL
LIN {X 0,Y 451.536,Z 479.365,A -85,B 0,C 180,E1 19945.643,E2 19945.643} C_VEL
LIN {X 0,Y 450.994,Z 490.635,A -85,B 0,C 180,E1 19945.325,E2 19945.325} C_VEL
LIN {X 0,Y 449.783,Z 498.204,A -85,B 0,C 180,E1 19945.163,E2 19945.163} C_VEL
LIN {X 0,Y 443.547,Z 517.242,A -85,B 0,C 180,E1 19944.878,E2 19944.878} C_VEL
LIN {X 0,Y 442.056,Z 524.493,A -85,B 0,C 180,E1 19944.611,E2 19944.611} C_VEL
LIN {X 0,Y 439.885,Z 544.43,A -85,B 0,C 180,E1 19943.497,E2 19943.497} C_VEL
LIN {X 0,Y 437.404,Z 563.728,A -85,B 0,C 180,E1 19942.165,E2 19942.165} C_VEL
LIN {X 0,Y 434.609,Z 582.464,A -85,B 0,C 180,E1 19940.582,E2 19940.582} C_VEL
LIN {X 0,Y 431.73,Z 599.884,A -85,B 0,C 180,E1 19938.824,E2 19938.824} C_VEL
LIN {X 0,Y 428.782,Z 617.004,A -85,B 0,C 180,E1 19936.778,E2 19936.778} C_VEL
LIN {X 0,Y 426.135,Z 631.875,A -85,B 0,C 180,E1 19934.688,E2 19934.688} C_VEL
LIN {X 0,Y 423.553,Z 646.334,A -85,B 0,C 180,E1 19932.283,E2 19932.283} C_VEL
LIN {X 0,Y 421.325,Z 659.216,A -85,B 0,C 180,E1 19929.744,E2 19929.744} C_VEL
LIN {X 0,Y 419.408,Z 671.209,A -85,B 0,C 180,E1 19926.925,E2 19926.925} C_VEL
LIN {X 0,Y 418.03,Z 681.047,A -85,B 0,C 180,E1 19924.149,E2 19924.149} C_VEL
LIN {X 0,Y 417.007,Z 689.723,A -85,B 0,C 180,E1 19921.131,E2 19921.131} C_VEL
LIN {X 0,Y 416.436,Z 695.931,A -85,B 0,C 180,E1 19918.385,E2 19918.385} C_VEL
LIN {X 0,Y 416.113,Z 701.276,A -85,B 0,C 180,E1 19915.322,E2 19915.322} C_VEL
LIN {X 0,Y 415.991,Z 704.674,A -85,B 0,C 180,E1 19912.468,E2 19912.468} C_VEL
LIN {X 0,Y 415.94,Z 706.663,A -85,B 0,C 180,E1 19909.666,E2 19909.666} C_VEL
LIN {X 0,Y 415.936,Z 707.257,A -85,B 0,C 180,E1 19906.479,E2 19906.479} C_VEL
LIN {X 0,Y 415.952,Z 706.387,A -85,B 0,C 180,E1 19903.767,E2 19903.767} C_VEL
LIN {X 0,Y 415.993,Z 704.046,A -85,B 0,C 180,E1 19900.806,E2 19900.806} C_VEL
LIN {X 0,Y 416.176,Z 699.91,A -85,B 0,C 180,E1 19897.732,E2 19897.732} C_VEL
LIN {X 0,Y 416.522,Z 694.779,A -85,B 0,C 180,E1 19894.987,E2 19894.987} C_VEL
LIN {X 0,Y 417.236,Z 687.355,A -85,B 0,C 180,E1 19891.923,E2 19891.923} C_VEL
LIN {X 0,Y 418.313,Z 678.584,A -85,B 0,C 180,E1 19889.042,E2 19889.042} C_VEL
LIN {X 0,Y 419.888,Z 667.965,A -85,B 0,C 180,E1 19886.177,E2 19886.177} C_VEL
LIN {X 0,Y 421.741,Z 656.425,A -85,B 0,C 180,E1 19883.603,E2 19883.603} C_VEL
LIN {X 0,Y 424.024,Z 643.329,A -85,B 0,C 180,E1 19881.123,E2 19881.123} C_VEL
LIN {X 0,Y 426.479,Z 629.75,A -85,B 0,C 180,E1 19878.916,E2 19878.916} C_VEL
LIN {X 0,Y 429.217,Z 614.415,A -85,B 0,C 180,E1 19876.804,E2 19876.804} C_VEL
LIN {X 0,Y 432,Z 598.198,A -85,B 0,C 180,E1 19874.908,E2 19874.908} C_VEL
LIN {X 0,Y 434.89,Z 580.614,A -85,B 0,C 180,E1 19873.161,E2 19873.161} C_VEL
LIN {X 0,Y 437.642,Z 562.185,A -85,B 0,C 180,E1 19871.622,E2 19871.622} C_VEL
LIN {X 0,Y 440.163,Z 542.52,A -85,B 0,C 180,E1 19870.286,E2 19870.286} C_VEL
LIN {X 0,Y 442.283,Z 522.988,A -85,B 0,C 180,E1 19869.211,E2 19869.211} C_VEL
LIN {X 0,Y 444.048,Z 503.078,A -85,B 0,C 180,E1 19868.342,E2 19868.342} C_VEL
LIN {X 0,Y 445.344,Z 482.178,A -85,B 0,C 180,E1 19867.663,E2 19867.663} C_VEL
LIN {X 0,Y 446.698,Z 448.531,A -85,B 0,C 180,E1 19866.948,E2 19866.948} C_VEL
LIN {X 0,Y 453.7,Z 272.593,A -85,B 0,C 180,E1 19863.555,E2 19863.555} C_VEL
LIN {X 0,Y 454.603,Z 244.025,A -85,B 0,C 180,E1 19863.005,E2 19863.005} C_VEL
LIN {X 0,Y 442.61,Z 226.303,A -85,B 0,C 180,E1 19861.113,E2 19861.113} C_VEL
LIN {X 0,Y 428.062,Z 209.169,A -85,B 0,C 180,E1 19858.749,E2 19858.749} C_VEL
LIN {X 0,Y 426.872,Z 207.757,A -85,B 0,C 180,E1 19858.496,E2 19858.496} C_VEL
LIN {X 0,Y 424.996,Z 204.125,A -85,B 0,C 180,E1 19857.63,E2 19857.63} C_VEL
LIN {X 0,Y 422.416,Z 199.37,A -85,B 0,C 180,E1 19856.428,E2 19856.428} C_VEL
LIN {X 0,Y 420.455,Z 196.053,A -85,B 0,C 180,E1 19855.53,E2 19855.53} C_VEL
LIN {X 0,Y 419.674,Z 194.452,A -85,B 0,C 180,E1 19855.125,E2 19855.125} C_VEL
LIN {X 0,Y 417.587,Z 191.011,A -85,B 0,C 180,E1 19854.145,E2 19854.145} C_VEL
LIN {X 0,Y 417.318,Z 189.748,A -85,B 0,C 180,E1 19853.846,E2 19853.846} C_VEL
LIN {X 0,Y 417.345,Z 189.75,A -85,B 0,C 180,E1 19849.875,E2 19849.875} C_VEL
LIN {X 0,Y 417.368,Z 189.741,A -85,B 0,C 180,E1 19845.947,E2 19845.947} C_VEL
LIN {X 0,Y 417.38,Z 189.739,A -85,B 0,C 180,E1 19842.045,E2 19842.045} C_VEL
LIN {X 0,Y 417.368,Z 189.744,A -85,B 0,C 180,E1 19838.176,E2 19838.176} C_VEL
LIN {X 0,Y 417.353,Z 189.749,A -85,B 0,C 180,E1 19834.43,E2 19834.43} C_VEL
LIN {X 0,Y 417.366,Z 189.74,A -85,B 0,C 180,E1 19830.523,E2 19830.523} C_VEL
LIN {X 0,Y 417.379,Z 189.728,A -85,B 0,C 180,E1 19826.678,E2 19826.678} C_VEL
LIN {X 0,Y 417.38,Z 189.721,A -85,B 0,C 180,E1 19822.737,E2 19822.737} C_VEL
LIN {X 0,Y 417.365,Z 189.731,A -85,B 0,C 180,E1 19818.866,E2 19818.866} C_VEL
LIN {X 0,Y 417.337,Z 189.749,A -85,B 0,C 180,E1 19815.092,E2 19815.092} C_VEL
LIN {X 0,Y 417.337,Z 189.75,A -85,B 0,C 180,E1 19811.19,E2 19811.19} C_VEL
LIN {X 0,Y 417.354,Z 189.739,A -85,B 0,C 180,E1 19807.434,E2 19807.434} C_VEL
LIN {X 0,Y 417.371,Z 189.727,A -85,B 0,C 180,E1 19803.572,E2 19803.572} C_VEL
LIN {X 0,Y 417.374,Z 189.727,A -85,B 0,C 180,E1 19799.726,E2 19799.726} C_VEL
LIN {X 0,Y 417.351,Z 189.73,A -85,B 0,C 180,E1 19795.879,E2 19795.879} C_VEL
LIN {X 0,Y 417.341,Z 189.732,A -85,B 0,C 180,E1 19792.152,E2 19792.152} C_VEL
LIN {X 0,Y 417.369,Z 189.729,A -85,B 0,C 180,E1 19788.391,E2 19788.391} C_VEL
LIN {X 0,Y 417.381,Z 189.729,A -85,B 0,C 180,E1 19784.58,E2 19784.58} C_VEL
LIN {X 0,Y 417.394,Z 189.912,A -85,B 0,C 180,E1 19784.117,E2 19784.117} C_VEL
LIN {X 0,Y 418.678,Z 193.223,A -85,B 0,C 180,E1 19783.347,E2 19783.347} C_VEL
LIN {X 0,Y 420.271,Z 195.341,A -85,B 0,C 180,E1 19782.7,E2 19782.7} C_VEL
LIN {X 0,Y 422.174,Z 199.058,A -85,B 0,C 180,E1 19781.783,E2 19781.783} C_VEL
LIN {X 0,Y 423.304,Z 201.16,A -85,B 0,C 180,E1 19781.263,E2 19781.263} C_VEL
LIN {X 0,Y 425.923,Z 205.967,A -85,B 0,C 180,E1 19780.1,E2 19780.1} C_VEL
LIN {X 0,Y 430.701,Z 214.971,A -85,B 0,C 180,E1 19778.053,E2 19778.053} C_VEL
LIN {X 0,Y 436.871,Z 227.089,A -85,B 0,C 180,E1 19775.528,E2 19775.528} C_VEL
LIN {X 0,Y 444.481,Z 243.043,A -85,B 0,C 180,E1 19772.539,E2 19772.539} C_VEL
LIN {X 0,Y 452.775,Z 261.702,A -85,B 0,C 180,E1 19769.402,E2 19769.402} C_VEL
LIN {X 0,Y 449.496,Z 292.756,A -85,B 0,C 180,E1 19766.673,E2 19766.673} C_VEL
LIN {X 0,Y 447.538,Z 318.099,A -85,B 0,C 180,E1 19764.412,E2 19764.412} C_VEL
LIN {X 0,Y 448.039,Z 336.895,A -85,B 0,C 180,E1 19762.555,E2 19762.555} C_VEL
LIN {X 0,Y 450.443,Z 353.393,A -85,B 0,C 180,E1 19760.757,E2 19760.757} C_VEL
LIN {X 0,Y 454.673,Z 368.482,A -85,B 0,C 180,E1 19758.963,E2 19758.963} C_VEL
LIN {X 0,Y 460.769,Z 382.243,A -85,B 0,C 180,E1 19757.177,E2 19757.177} C_VEL
LIN {X 0,Y 468.151,Z 393.861,A -85,B 0,C 180,E1 19755.531,E2 19755.531} C_VEL
LIN {X 0,Y 477.893,Z 405.051,A -85,B 0,C 180,E1 19753.796,E2 19753.796} C_VEL
LIN {X 0,Y 482.811,Z 409.639,A -85,B 0,C 180,E1 19753.037,E2 19753.037} C_VEL
LIN {X 0,Y 472.959,Z 425.816,A -85,B 0,C 180,E1 19752.479,E2 19752.479} C_VEL
LIN {X 0,Y 467.76,Z 435.017,A -85,B 0,C 180,E1 19752.122,E2 19752.122} C_VEL
LIN {X 0,Y 458.658,Z 450.795,A -85,B 0,C 180,E1 19751.507,E2 19751.507} C_VEL
LIN {X 0,Y 452.309,Z 464.71,A -85,B 0,C 180,E1 19750.853,E2 19750.853} C_VEL
LIN {X 0,Y 449.765,Z 482.199,A -85,B 0,C 180,E1 19750.765,E2 19750.765} C_VEL
LIN {X 0,Y 448.474,Z 498.965,A -85,B 0,C 180,E1 19750.549,E2 19750.549} C_VEL
LIN {X 0,Y 446.921,Z 525.019,A -85,B 0,C 180,E1 19749.958,E2 19749.958} C_VEL
LIN {X 0,Y 444.465,Z 549.728,A -85,B 0,C 180,E1 19749.181,E2 19749.181} C_VEL
LIN {X 0,Y 441.753,Z 573.805,A -85,B 0,C 180,E1 19748.163,E2 19748.163} C_VEL
LIN {X 0,Y 438.951,Z 596.145,A -85,B 0,C 180,E1 19746.966,E2 19746.966} C_VEL
LIN {X 0,Y 436.053,Z 617.837,A -85,B 0,C 180,E1 19745.54,E2 19745.54} C_VEL
LIN {X 0,Y 433.109,Z 638.382,A -85,B 0,C 180,E1 19743.909,E2 19743.909} C_VEL
LIN {X 0,Y 430.122,Z 658.453,A -85,B 0,C 180,E1 19742.006,E2 19742.006} C_VEL
LIN {X 0,Y 427.253,Z 677.223,A -85,B 0,C 180,E1 19739.898,E2 19739.898} C_VEL
LIN {X 0,Y 424.502,Z 695.207,A -85,B 0,C 180,E1 19737.494,E2 19737.494} C_VEL
LIN {X 0,Y 422.227,Z 710.503,A -85,B 0,C 180,E1 19735.08,E2 19735.08} C_VEL
LIN {X 0,Y 420.295,Z 724.352,A -85,B 0,C 180,E1 19732.52,E2 19732.52} C_VEL
LIN {X 0,Y 418.668,Z 737.298,A -85,B 0,C 180,E1 19729.678,E2 19729.678} C_VEL
LIN {X 0,Y 417.44,Z 748.655,A -85,B 0,C 180,E1 19726.649,E2 19726.649} C_VEL
LIN {X 0,Y 416.703,Z 757.087,A -85,B 0,C 180,E1 19723.883,E2 19723.883} C_VEL
LIN {X 0,Y 416.257,Z 764.013,A -85,B 0,C 180,E1 19721.079,E2 19721.079} C_VEL
LIN {X 0,Y 416.029,Z 769.664,A -85,B 0,C 180,E1 19718.013,E2 19718.013} C_VEL
LIN {X 0,Y 415.953,Z 773.194,A -85,B 0,C 180,E1 19715.241,E2 19715.241} C_VEL
LIN {X 0,Y 415.934,Z 775.309,A -85,B 0,C 180,E1 19712.342,E2 19712.342} C_VEL
LIN {X 0,Y 415.925,Z 775.797,A -85,B 0,C 180,E1 19709.587,E2 19709.587} C_VEL
LIN {X 0,Y 415.937,Z 774.779,A -85,B 0,C 180,E1 19706.692,E2 19706.692} C_VEL
LIN {X 0,Y 415.964,Z 772.097,A -85,B 0,C 180,E1 19703.79,E2 19703.79} C_VEL
LIN {X 0,Y 416.086,Z 767.757,A -85,B 0,C 180,E1 19700.874,E2 19700.874} C_VEL
LIN {X 0,Y 416.385,Z 761.659,A -85,B 0,C 180,E1 19697.941,E2 19697.941} C_VEL
LIN {X 0,Y 416.957,Z 753.666,A -85,B 0,C 180,E1 19694.99,E2 19694.99} C_VEL
LIN {X 0,Y 417.847,Z 744.148,A -85,B 0,C 180,E1 19692.164,E2 19692.164} C_VEL
LIN {X 0,Y 419.153,Z 732.515,A -85,B 0,C 180,E1 19689.326,E2 19689.326} C_VEL
LIN {X 0,Y 420.938,Z 718.48,A -85,B 0,C 180,E1 19686.481,E2 19686.481} C_VEL
LIN {X 0,Y 423.011,Z 703.418,A -85,B 0,C 180,E1 19683.919,E2 19683.919} C_VEL
LIN {X 0,Y 425.387,Z 686.872,A -85,B 0,C 180,E1 19681.53,E2 19681.53} C_VEL
LIN {X 0,Y 428.055,Z 668.741,A -85,B 0,C 180,E1 19679.311,E2 19679.311} C_VEL
LIN {X 0,Y 430.788,Z 649.626,A -85,B 0,C 180,E1 19677.341,E2 19677.341} C_VEL
LIN {X 0,Y 433.453,Z 630.684,A -85,B 0,C 180,E1 19675.67,E2 19675.67} C_VEL
LIN {X 0,Y 436.341,Z 609.21,A -85,B 0,C 180,E1 19674.083,E2 19674.083} C_VEL
LIN {X 0,Y 439.189,Z 587.36,A -85,B 0,C 180,E1 19672.729,E2 19672.729} C_VEL
LIN {X 0,Y 441.951,Z 563.92,A -85,B 0,C 180,E1 19671.567,E2 19671.567} C_VEL
LIN {X 0,Y 444.689,Z 539.036,A -85,B 0,C 180,E1 19670.613,E2 19670.613} C_VEL
LIN {X 0,Y 446.968,Z 513.71,A -85,B 0,C 180,E1 19669.885,E2 19669.885} C_VEL
LIN {X 0,Y 448.312,Z 489.422,A -85,B 0,C 180,E1 19669.385,E2 19669.385} C_VEL
LIN {X 0,Y 450.428,Z 465.325,A -85,B 0,C 180,E1 19669.126,E2 19669.126} C_VEL
LIN {X 0,Y 451.599,Z 454.302,A -85,B 0,C 180,E1 19669.011,E2 19669.011} C_VEL
LIN {X 0,Y 457.978,Z 434.515,A -85,B 0,C 180,E1 19668.334,E2 19668.334} C_VEL
LIN {X 0,Y 461.803,Z 423.847,A -85,B 0,C 180,E1 19668.008,E2 19668.008} C_VEL
LIN {X 0,Y 468.18,Z 404.709,A -85,B 0,C 180,E1 19667.39,E2 19667.39} C_VEL
LIN {X 0,Y 477.741,Z 381.434,A -85,B 0,C 180,E1 19666.813,E2 19666.813} C_VEL
LIN {X 0,Y 491.813,Z 351.818,A -85,B 0,C 180,E1 19666.273,E2 19666.273} C_VEL
LIN {X 0,Y 497.053,Z 341.141,A -85,B 0,C 180,E1 19666.097,E2 19666.097} C_VEL
LIN {X 0,Y 502.277,Z 326.453,A -85,B 0,C 180,E1 19665.691,E2 19665.691} C_VEL
LIN {X 0,Y 488.54,Z 315.374,A -85,B 0,C 180,E1 19663.769,E2 19663.769} C_VEL
LIN {X 0,Y 478.88,Z 304.527,A -85,B 0,C 180,E1 19662.084,E2 19662.084} C_VEL
LIN {X 0,Y 471.918,Z 293.828,A -85,B 0,C 180,E1 19660.575,E2 19660.575} C_VEL
LIN {X 0,Y 464.688,Z 277.769,A -85,B 0,C 180,E1 19658.529,E2 19658.529} C_VEL
LIN {X 0,Y 457.84,Z 260.876,A -85,B 0,C 180,E1 19656.286,E2 19656.286} C_VEL
LIN {X 0,Y 455.263,Z 255.593,A -85,B 0,C 180,E1 19655.475,E2 19655.475} C_VEL
LIN {X 0,Y 451.991,Z 257.309,A -85,B 0,C 180,E1 19655.11,E2 19655.11} C_VEL
LIN {X 0,Y 447.283,Z 260.161,A -85,B 0,C 180,E1 19654.596,E2 19654.596} C_VEL
LIN {X 0,Y 445.785,Z 260.927,A -85,B 0,C 180,E1 19654.417,E2 19654.417} C_VEL
LIN {X 0,Y 441.779,Z 263.655,A -85,B 0,C 180,E1 19653.988,E2 19653.988} C_VEL
LIN {X 0,Y 439.266,Z 264.763,A -85,B 0,C 180,E1 19653.659,E2 19653.659} C_VEL
LIN {X 0,Y 435.59,Z 267.532,A -85,B 0,C 180,E1 19653.271,E2 19653.271} C_VEL
LIN {X 0,Y 432.98,Z 268.326,A -85,B 0,C 180,E1 19652.847,E2 19652.847} C_VEL
LIN {X 0,Y 432.24,Z 307.579,A -85,B 0,C 180,E1 19649.442,E2 19649.442} C_VEL
LIN {X 0,Y 431.346,Z 340.693,A -85,B 0,C 180,E1 19646.501,E2 19646.501} C_VEL
LIN {X 0,Y 429.369,Z 349.299,A -85,B 0,C 180,E1 19645.949,E2 19645.949} C_VEL
LIN {X 0,Y 425.809,Z 452.457,A -85,B 0,C 180,E1 19643.641,E2 19643.641} C_VEL
LIN {X 0,Y 424.915,Z 506.45,A -85,B 0,C 180,E1 19642.519,E2 19642.519} C_VEL
LIN {X 0,Y 424.865,Z 524.271,A -85,B 0,C 180,E1 19641.99,E2 19641.99} C_VEL
LIN {X 0,Y 424.565,Z 541.448,A -85,B 0,C 180,E1 19641.228,E2 19641.228} C_VEL
LIN {X 0,Y 424.075,Z 557.294,A -85,B 0,C 180,E1 19640.278,E2 19640.278} C_VEL
LIN {X 0,Y 423.385,Z 572.524,A -85,B 0,C 180,E1 19639.091,E2 19639.091} C_VEL
LIN {X 0,Y 422.582,Z 586.585,A -85,B 0,C 180,E1 19637.712,E2 19637.712} C_VEL
LIN {X 0,Y 421.753,Z 598.783,A -85,B 0,C 180,E1 19636.23,E2 19636.23} C_VEL
LIN {X 0,Y 420.895,Z 609.767,A -85,B 0,C 180,E1 19634.584,E2 19634.584} C_VEL
LIN {X 0,Y 420.022,Z 620.14,A -85,B 0,C 180,E1 19632.65,E2 19632.65} C_VEL
LIN {X 0,Y 419.317,Z 628.36,A -85,B 0,C 180,E1 19630.718,E2 19630.718} C_VEL
LIN {X 0,Y 418.709,Z 635.124,A -85,B 0,C 180,E1 19628.652,E2 19628.652} C_VEL
LIN {X 0,Y 418.212,Z 640.391,A -85,B 0,C 180,E1 19626.451,E2 19626.451} C_VEL
LIN {X 0,Y 417.874,Z 643.878,A -85,B 0,C 180,E1 19624.253,E2 19624.253} C_VEL
LIN {X 0,Y 417.663,Z 645.722,A -85,B 0,C 180,E1 19622.057,E2 19622.057} C_VEL
LIN {X 0,Y 417.533,Z 645.884,A -85,B 0,C 180,E1 19619.725,E2 19619.725} C_VEL
LIN {X 0,Y 417.493,Z 644.281,A -85,B 0,C 180,E1 19617.391,E2 19617.391} C_VEL
LIN {X 0,Y 417.577,Z 640.912,A -85,B 0,C 180,E1 19615.055,E2 19615.055} C_VEL
LIN {X 0,Y 417.795,Z 635.586,A -85,B 0,C 180,E1 19612.713,E2 19612.713} C_VEL
LIN {X 0,Y 418.171,Z 628.697,A -85,B 0,C 180,E1 19610.503,E2 19610.503} C_VEL
LIN {X 0,Y 418.682,Z 620.337,A -85,B 0,C 180,E1 19608.427,E2 19608.427} C_VEL
LIN {X 0,Y 419.332,Z 610.489,A -85,B 0,C 180,E1 19606.486,E2 19606.486} C_VEL
LIN {X 0,Y 420.179,Z 598.295,A -85,B 0,C 180,E1 19604.542,E2 19604.542} C_VEL
LIN {X 0,Y 421.052,Z 585.385,A -85,B 0,C 180,E1 19602.874,E2 19602.874} C_VEL
LIN {X 0,Y 421.963,Z 570.714,A -85,B 0,C 180,E1 19601.343,E2 19601.343} C_VEL
LIN {X 0,Y 422.832,Z 554.973,A -85,B 0,C 180,E1 19600.022,E2 19600.022} C_VEL
LIN {X 0,Y 423.54,Z 538.964,A -85,B 0,C 180,E1 19598.971,E2 19598.971} C_VEL
LIN {X 0,Y 424.127,Z 520.953,A -85,B 0,C 180,E1 19598.082,E2 19598.082} C_VEL
LIN {X 0,Y 424.497,Z 503.12,A -85,B 0,C 180,E1 19597.468,E2 19597.468} C_VEL
LIN {X 0,Y 425.081,Z 459.582,A -85,B 0,C 180,E1 19596.599,E2 19596.599} C_VEL
LIN {X 0,Y 427.688,Z 335.939,A -85,B 0,C 180,E1 19594.176,E2 19594.176} C_VEL
LIN {X 0,Y 426.907,Z 330.377,A -85,B 0,C 180,E1 19593.988,E2 19593.988} C_VEL
LIN {X 0,Y 427.402,Z 319.252,A -85,B 0,C 180,E1 19592.877,E2 19592.877} C_VEL
LIN {X 0,Y 428.692,Z 320.308,A -85,B 0,C 180,E1 19592.646,E2 19592.646} C_VEL
LIN {X 0,Y 431.123,Z 319.776,A -85,B 0,C 180,E1 19592.289,E2 19592.289} C_VEL
LIN {X 0,Y 434.681,Z 316.677,A -85,B 0,C 180,E1 19591.846,E2 19591.846} C_VEL
LIN {X 0,Y 436.209,Z 314.92,A -85,B 0,C 180,E1 19591.674,E2 19591.674} C_VEL
LIN {X 0,Y 439.807,Z 314.033,A -85,B 0,C 180,E1 19591.186,E2 19591.186} C_VEL
LIN {X 0,Y 444.081,Z 310.938,A -85,B 0,C 180,E1 19590.678,E2 19590.678} C_VEL
LIN {X 0,Y 445.807,Z 309.574,A -85,B 0,C 180,E1 19590.484,E2 19590.484} C_VEL
LIN {X 0,Y 450.622,Z 307.618,A -85,B 0,C 180,E1 19589.903,E2 19589.903} C_VEL
LIN {X 0,Y 452.376,Z 306.664,A -85,B 0,C 180,E1 19589.702,E2 19589.702} C_VEL
LIN {X 0,Y 445.145,Z 481.091,A -85,B 0,C 180,E1 19586.233,E2 19586.233} C_VEL
LIN {X 0,Y 443.953,Z 501.957,A -85,B 0,C 180,E1 19585.581,E2 19585.581} C_VEL
LIN {X 0,Y 442.248,Z 522.601,A -85,B 0,C 180,E1 19584.704,E2 19584.704} C_VEL
LIN {X 0,Y 442.056,Z 524.493,A -85,B 0,C 180,E1 19584.611,E2 19584.611} C_VEL
LIN {X 0,Y 440.526,Z 531.827,A -85,B 0,C 180,E1 19584.317,E2 19584.317} C_VEL
LIN {X 0,Y 433.627,Z 550.086,A -85,B 0,C 180,E1 19583.714,E2 19583.714} C_VEL
LIN {X 0,Y 431.864,Z 556.99,A -85,B 0,C 180,E1 19583.314,E2 19583.314} C_VEL
LIN {X 0,Y 429.125,Z 575.385,A -85,B 0,C 180,E1 19581.869,E2 19581.869} C_VEL
LIN {X 0,Y 426.067,Z 593.754,A -85,B 0,C 180,E1 19580.119,E2 19580.119} C_VEL
LIN {X 0,Y 423.014,Z 610.719,A -85,B 0,C 180,E1 19578.198,E2 19578.198} C_VEL
LIN {X 0,Y 419.869,Z 627.458,A -85,B 0,C 180,E1 19575.944,E2 19575.944} C_VEL
LIN {X 0,Y 417.098,Z 642.096,A -85,B 0,C 180,E1 19573.618,E2 19573.618} C_VEL
LIN {X 0,Y 414.595,Z 655.61,A -85,B 0,C 180,E1 19571.079,E2 19571.079} C_VEL
LIN {X 0,Y 412.446,Z 667.705,A -85,B 0,C 180,E1 19568.36,E2 19568.36} C_VEL
LIN {X 0,Y 410.789,Z 678.078,A -85,B 0,C 180,E1 19565.572,E2 19565.572} C_VEL
LIN {X 0,Y 409.547,Z 687.149,A -85,B 0,C 180,E1 19562.618,E2 19562.618} C_VEL
LIN {X 0,Y 408.727,Z 694.572,A -85,B 0,C 180,E1 19559.614,E2 19559.614} C_VEL
LIN {X 0,Y 408.279,Z 700.167,A -85,B 0,C 180,E1 19556.626,E2 19556.626} C_VEL
LIN {X 0,Y 408.052,Z 704.37,A -85,B 0,C 180,E1 19553.541,E2 19553.541} C_VEL
LIN {X 0,Y 407.98,Z 706.911,A -85,B 0,C 180,E1 19550.516,E2 19550.516} C_VEL
LIN {X 0,Y 407.961,Z 707.883,A -85,B 0,C 180,E1 19547.693,E2 19547.693} C_VEL
LIN {X 0,Y 407.976,Z 707.447,A -85,B 0,C 180,E1 19544.518,E2 19544.518} C_VEL
LIN {X 0,Y 408.013,Z 705.556,A -85,B 0,C 180,E1 19541.593,E2 19541.593} C_VEL
LIN {X 0,Y 408.145,Z 702.111,A -85,B 0,C 180,E1 19538.594,E2 19538.594} C_VEL
LIN {X 0,Y 408.505,Z 696.872,A -85,B 0,C 180,E1 19535.478,E2 19535.478} C_VEL
LIN {X 0,Y 409.156,Z 690.341,A -85,B 0,C 180,E1 19532.521,E2 19532.521} C_VEL
LIN {X 0,Y 410.179,Z 682.026,A -85,B 0,C 180,E1 19529.581,E2 19529.581} C_VEL
LIN {X 0,Y 411.612,Z 672.445,A -85,B 0,C 180,E1 19526.797,E2 19526.797} C_VEL
LIN {X 0,Y 413.448,Z 661.71,A -85,B 0,C 180,E1 19524.171,E2 19524.171} C_VEL
LIN {X 0,Y 415.739,Z 649.005,A -85,B 0,C 180,E1 19521.564,E2 19521.564} C_VEL
LIN {X 0,Y 418.244,Z 635.676,A -85,B 0,C 180,E1 19519.253,E2 19519.253} C_VEL
LIN {X 0,Y 421.174,Z 620.223,A -85,B 0,C 180,E1 19516.966,E2 19516.966} C_VEL
LIN {X 0,Y 424.123,Z 604.396,A -85,B 0,C 180,E1 19514.97,E2 19514.97} C_VEL
LIN {X 0,Y 427.136,Z 586.906,A -85,B 0,C 180,E1 19513.126,E2 19513.126} C_VEL
LIN {X 0,Y 429.952,Z 569.283,A -85,B 0,C 180,E1 19511.563,E2 19511.563} C_VEL
LIN {X 0,Y 432.565,Z 551.131,A -85,B 0,C 180,E1 19510.207,E2 19510.207} C_VEL
LIN {X 0,Y 434.857,Z 532.235,A -85,B 0,C 180,E1 19509.051,E2 19509.051} C_VEL
LIN {X 0,Y 436.87,Z 511.95,A -85,B 0,C 180,E1 19508.069,E2 19508.069} C_VEL
LIN {X 0,Y 438.478,Z 490.605,A -85,B 0,C 180,E1 19507.285,E2 19507.285} C_VEL
LIN {X 0,Y 439.499,Z 469.99,A -85,B 0,C 180,E1 19506.746,E2 19506.746} C_VEL
LIN {X 0,Y 447.212,Z 288.193,A -85,B 0,C 180,E1 19503.156,E2 19503.156} C_VEL
LIN {X 0,Y 448.66,Z 247.56,A -85,B 0,C 180,E1 19502.371,E2 19502.371} C_VEL
LIN {X 0,Y 438.283,Z 232.287,A -85,B 0,C 180,E1 19500.697,E2 19500.697} C_VEL
LIN {X 0,Y 424.243,Z 215.604,A -85,B 0,C 180,E1 19498.365,E2 19498.365} C_VEL
LIN {X 0,Y 420.451,Z 210.951,A -85,B 0,C 180,E1 19497.652,E2 19497.652} C_VEL
LIN {X 0,Y 416.882,Z 204.804,A -85,B 0,C 180,E1 19496.025,E2 19496.025} C_VEL
LIN {X 0,Y 414.522,Z 200.391,A -85,B 0,C 180,E1 19494.856,E2 19494.856} C_VEL
LIN {X 0,Y 412.47,Z 196.71,A -85,B 0,C 180,E1 19493.826,E2 19493.826} C_VEL
LIN {X 0,Y 411.794,Z 195.53,A -85,B 0,C 180,E1 19493.485,E2 19493.485} C_VEL
LIN {X 0,Y 409.744,Z 192.229,A -85,B 0,C 180,E1 19492.474,E2 19492.474} C_VEL
LIN {X 0,Y 409.39,Z 190.723,A -85,B 0,C 180,E1 19492.081,E2 19492.081} C_VEL
LIN {X 0,Y 409.419,Z 190.718,A -85,B 0,C 180,E1 19488.358,E2 19488.358} C_VEL
LIN {X 0,Y 409.435,Z 190.714,A -85,B 0,C 180,E1 19484.497,E2 19484.497} C_VEL
LIN {X 0,Y 409.447,Z 190.711,A -85,B 0,C 180,E1 19480.51,E2 19480.51} C_VEL
LIN {X 0,Y 409.428,Z 190.715,A -85,B 0,C 180,E1 19476.75,E2 19476.75} C_VEL
LIN {X 0,Y 409.417,Z 190.719,A -85,B 0,C 180,E1 19472.831,E2 19472.831} C_VEL
LIN {X 0,Y 409.447,Z 190.726,A -85,B 0,C 180,E1 19468.916,E2 19468.916} C_VEL
LIN {X 0,Y 409.442,Z 190.734,A -85,B 0,C 180,E1 19464.991,E2 19464.991} C_VEL
LIN {X 0,Y 409.429,Z 190.733,A -85,B 0,C 180,E1 19461.038,E2 19461.038} C_VEL
LIN {X 0,Y 409.405,Z 190.722,A -85,B 0,C 180,E1 19457.189,E2 19457.189} C_VEL
LIN {X 0,Y 409.377,Z 190.718,A -85,B 0,C 180,E1 19453.417,E2 19453.417} C_VEL
LIN {X 0,Y 409.398,Z 190.723,A -85,B 0,C 180,E1 19449.56,E2 19449.56} C_VEL
LIN {X 0,Y 409.422,Z 190.731,A -85,B 0,C 180,E1 19445.747,E2 19445.747} C_VEL
LIN {X 0,Y 409.439,Z 190.736,A -85,B 0,C 180,E1 19441.82,E2 19441.82} C_VEL
LIN {X 0,Y 409.432,Z 190.737,A -85,B 0,C 180,E1 19437.901,E2 19437.901} C_VEL
LIN {X 0,Y 409.402,Z 190.74,A -85,B 0,C 180,E1 19433.972,E2 19433.972} C_VEL
LIN {X 0,Y 409.412,Z 190.738,A -85,B 0,C 180,E1 19430.157,E2 19430.157} C_VEL
LIN {X 0,Y 409.435,Z 190.736,A -85,B 0,C 180,E1 19426.298,E2 19426.298} C_VEL
LIN {X 0,Y 409.446,Z 190.924,A -85,B 0,C 180,E1 19425.826,E2 19425.826} C_VEL
LIN {X 0,Y 410.66,Z 194.066,A -85,B 0,C 180,E1 19425.044,E2 19425.044} C_VEL
LIN {X 0,Y 412.28,Z 195.905,A -85,B 0,C 180,E1 19424.384,E2 19424.384} C_VEL
LIN {X 0,Y 413.966,Z 199.682,A -85,B 0,C 180,E1 19423.441,E2 19423.441} C_VEL
LIN {X 0,Y 415.202,Z 201.441,A -85,B 0,C 180,E1 19422.915,E2 19422.915} C_VEL
LIN {X 0,Y 417.461,Z 205.513,A -85,B 0,C 180,E1 19421.859,E2 19421.859} C_VEL
LIN {X 0,Y 423.488,Z 217.036,A -85,B 0,C 180,E1 19419.114,E2 19419.114} C_VEL
LIN {X 0,Y 429.822,Z 229.492,A -85,B 0,C 180,E1 19416.415,E2 19416.415} C_VEL
LIN {X 0,Y 437.016,Z 244.397,A -85,B 0,C 180,E1 19413.504,E2 19413.504} C_VEL
LIN {X 0,Y 445.355,Z 263.079,A -85,B 0,C 180,E1 19410.254,E2 19410.254} C_VEL
LIN {X 0,Y 446.505,Z 265.801,A -85,B 0,C 180,E1 19409.811,E2 19409.811} C_VEL
LIN {X 0,Y 441.066,Z 319.711,A -85,B 0,C 180,E1 19405.004,E2 19405.004} C_VEL
LIN {X 0,Y 441.345,Z 338.8,A -85,B 0,C 180,E1 19403.103,E2 19403.103} C_VEL
LIN {X 0,Y 443.561,Z 355.667,A -85,B 0,C 180,E1 19401.255,E2 19401.255} C_VEL
LIN {X 0,Y 447.587,Z 371.021,A -85,B 0,C 180,E1 19399.422,E2 19399.422} C_VEL
LIN {X 0,Y 453.295,Z 384.743,A -85,B 0,C 180,E1 19397.64,E2 19397.64} C_VEL
LIN {X 0,Y 460.356,Z 396.641,A -85,B 0,C 180,E1 19395.964,E2 19395.964} C_VEL
LIN {X 0,Y 469.842,Z 408.26,A -85,B 0,C 180,E1 19394.18,E2 19394.18} C_VEL
LIN {X 0,Y 473.866,Z 412.501,A -85,B 0,C 180,E1 19393.503,E2 19393.503} C_VEL
LIN {X 0,Y 464.698,Z 428.25,A -85,B 0,C 180,E1 19392.921,E2 19392.921} C_VEL
LIN {X 0,Y 452.928,Z 448.367,A -85,B 0,C 180,E1 19392.151,E2 19392.151} C_VEL
LIN {X 0,Y 446.525,Z 462.052,A -85,B 0,C 180,E1 19391.525,E2 19391.525} C_VEL
LIN {X 0,Y 443.613,Z 482.097,A -85,B 0,C 180,E1 19391.421,E2 19391.421} C_VEL
LIN {X 0,Y 442.251,Z 499.166,A -85,B 0,C 180,E1 19391.197,E2 19391.197} C_VEL
LIN {X 0,Y 440.562,Z 524.72,A -85,B 0,C 180,E1 19390.59,E2 19390.59} C_VEL
LIN {X 0,Y 437.946,Z 549.717,A -85,B 0,C 180,E1 19389.789,E2 19389.789} C_VEL
LIN {X 0,Y 435.133,Z 573.52,A -85,B 0,C 180,E1 19388.767,E2 19388.767} C_VEL
LIN {X 0,Y 432.206,Z 595.717,A -85,B 0,C 180,E1 19387.559,E2 19387.559} C_VEL
LIN {X 0,Y 429.054,Z 617.952,A -85,B 0,C 180,E1 19386.069,E2 19386.069} C_VEL
LIN {X 0,Y 425.961,Z 638.497,A -85,B 0,C 180,E1 19384.407,E2 19384.407} C_VEL
LIN {X 0,Y 422.92,Z 657.957,A -85,B 0,C 180,E1 19382.537,E2 19382.537} C_VEL
LIN {X 0,Y 420.003,Z 676.174,A -85,B 0,C 180,E1 19380.469,E2 19380.469} C_VEL
LIN {X 0,Y 417.022,Z 694.684,A -85,B 0,C 180,E1 19377.968,E2 19377.968} C_VEL
LIN {X 0,Y 414.53,Z 710.477,A -85,B 0,C 180,E1 19375.426,E2 19375.426} C_VEL
LIN {X 0,Y 412.492,Z 724.214,A -85,B 0,C 180,E1 19372.819,E2 19372.819} C_VEL
LIN {X 0,Y 410.846,Z 736.581,A -85,B 0,C 180,E1 19370.051,E2 19370.051} C_VEL
LIN {X 0,Y 409.556,Z 747.737,A -85,B 0,C 180,E1 19367.035,E2 19367.035} C_VEL
LIN {X 0,Y 408.757,Z 756.393,A -85,B 0,C 180,E1 19364.159,E2 19364.159} C_VEL
LIN {X 0,Y 408.286,Z 763.33,A -85,B 0,C 180,E1 19361.298,E2 19361.298} C_VEL
LIN {X 0,Y 408.044,Z 769.07,A -85,B 0,C 180,E1 19358.132,E2 19358.132} C_VEL
LIN {X 0,Y 407.972,Z 772.67,A -85,B 0,C 180,E1 19355.202,E2 19355.202} C_VEL
LIN {X 0,Y 407.959,Z 774.724,A -85,B 0,C 180,E1 19352.247,E2 19352.247} C_VEL
LIN {X 0,Y 407.954,Z 775.11,A -85,B 0,C 180,E1 19349.298,E2 19349.298} C_VEL
LIN {X 0,Y 407.959,Z 774.015,A -85,B 0,C 180,E1 19346.487,E2 19346.487} C_VEL
LIN {X 0,Y 407.986,Z 771.24,A -85,B 0,C 180,E1 19343.527,E2 19343.527} C_VEL
LIN {X 0,Y 408.123,Z 766.794,A -85,B 0,C 180,E1 19340.552,E2 19340.552} C_VEL
LIN {X 0,Y 408.442,Z 760.569,A -85,B 0,C 180,E1 19337.559,E2 19337.559} C_VEL
LIN {X 0,Y 409.033,Z 752.848,A -85,B 0,C 180,E1 19334.692,E2 19334.692} C_VEL
LIN {X 0,Y 409.978,Z 743.267,A -85,B 0,C 180,E1 19331.81,E2 19331.81} C_VEL
LIN {X 0,Y 411.369,Z 731.584,A -85,B 0,C 180,E1 19328.916,E2 19328.916} C_VEL
LIN {X 0,Y 413.163,Z 718.22,A -85,B 0,C 180,E1 19326.162,E2 19326.162} C_VEL
LIN {X 0,Y 415.321,Z 703.419,A -85,B 0,C 180,E1 19323.58,E2 19323.58} C_VEL
LIN {X 0,Y 417.877,Z 686.594,A -85,B 0,C 180,E1 19321.097,E2 19321.097} C_VEL
LIN {X 0,Y 420.737,Z 668.138,A -85,B 0,C 180,E1 19318.797,E2 19318.797} C_VEL
LIN {X 0,Y 423.535,Z 649.851,A -85,B 0,C 180,E1 19316.872,E2 19316.872} C_VEL
LIN {X 0,Y 426.447,Z 630.127,A -85,B 0,C 180,E1 19315.104,E2 19315.104} C_VEL
LIN {X 0,Y 429.65,Z 607.873,A -85,B 0,C 180,E1 19313.434,E2 19313.434} C_VEL
LIN {X 0,Y 432.628,Z 585.85,A -85,B 0,C 180,E1 19312.065,E2 19312.065} C_VEL
LIN {X 0,Y 435.503,Z 563.143,A -85,B 0,C 180,E1 19310.925,E2 19310.925} C_VEL
LIN {X 0,Y 438.372,Z 538.855,A -85,B 0,C 180,E1 19309.969,E2 19309.969} C_VEL
LIN {X 0,Y 440.832,Z 513.028,A -85,B 0,C 180,E1 19309.21,E2 19309.21} C_VEL
LIN {X 0,Y 442.299,Z 489.393,A -85,B 0,C 180,E1 19308.706,E2 19308.706} C_VEL
LIN {X 0,Y 444.492,Z 465.093,A -85,B 0,C 180,E1 19308.439,E2 19308.439} C_VEL
LIN {X 0,Y 446.024,Z 450.725,A -85,B 0,C 180,E1 19308.295,E2 19308.295} C_VEL
LIN {X 0,Y 452.64,Z 431.085,A -85,B 0,C 180,E1 19307.644,E2 19307.644} C_VEL
LIN {X 0,Y 455.957,Z 421.565,A -85,B 0,C 180,E1 19307.343,E2 19307.343} C_VEL
LIN {X 0,Y 462.944,Z 401.284,A -85,B 0,C 180,E1 19306.706,E2 19306.706} C_VEL
LIN {X 0,Y 472.843,Z 377.634,A -85,B 0,C 180,E1 19306.142,E2 19306.142} C_VEL
LIN {X 0,Y 487.439,Z 347.246,A -85,B 0,C 180,E1 19305.615,E2 19305.615} C_VEL
LIN {X 0,Y 491.262,Z 339.277,A -85,B 0,C 180,E1 19305.48,E2 19305.48} C_VEL
LIN {X 0,Y 494.34,Z 330.456,A -85,B 0,C 180,E1 19305.229,E2 19305.229} C_VEL
LIN {X 0,Y 482.76,Z 320.809,A -85,B 0,C 180,E1 19303.539,E2 19303.539} C_VEL
LIN {X 0,Y 472.932,Z 309.425,A -85,B 0,C 180,E1 19301.756,E2 19301.756} C_VEL
LIN {X 0,Y 466.092,Z 298.545,A -85,B 0,C 180,E1 19300.209,E2 19300.209} C_VEL
LIN {X 0,Y 458.69,Z 281.518,A -85,B 0,C 180,E1 19298.009,E2 19298.009} C_VEL
LIN {X 0,Y 452.35,Z 265.692,A -85,B 0,C 180,E1 19295.855,E2 19295.855} C_VEL
LIN {X 0,Y 451.707,Z 264.259,A -85,B 0,C 180,E1 19295.641,E2 19295.641} C_VEL
LIN {X 0,Y 445.168,Z 268.141,A -85,B 0,C 180,E1 19294.935,E2 19294.935} C_VEL
LIN {X 0,Y 440.52,Z 270.917,A -85,B 0,C 180,E1 19294.413,E2 19294.413} C_VEL
LIN {X 0,Y 438.979,Z 271.816,A -85,B 0,C 180,E1 19294.235,E2 19294.235} C_VEL
LIN {X 0,Y 435.014,Z 274.448,A -85,B 0,C 180,E1 19293.795,E2 19293.795} C_VEL
LIN {X 0,Y 432.883,Z 275.345,A -85,B 0,C 180,E1 19293.506,E2 19293.506} C_VEL
LIN {X 0,Y 429.527,Z 278.08,A -85,B 0,C 180,E1 19293.163,E2 19293.163} C_VEL
LIN {X 0,Y 426.813,Z 279.105,A -85,B 0,C 180,E1 19292.761,E2 19292.761} C_VEL
LIN {X 0,Y 426.532,Z 279.258,A -85,B 0,C 180,E1 19292.695,E2 19292.695} C_VEL
LIN {X 0,Y 425.433,Z 320.386,A -85,B 0,C 180,E1 19289.039,E2 19289.039} C_VEL
LIN {X 0,Y 424.572,Z 342.841,A -85,B 0,C 180,E1 19287.033,E2 19287.033} C_VEL
LIN {X 0,Y 422.558,Z 351.498,A -85,B 0,C 180,E1 19286.484,E2 19286.484} C_VEL
LIN {X 0,Y 418.8,Z 448.264,A -85,B 0,C 180,E1 19284.225,E2 19284.225} C_VEL
LIN {X 0,Y 417.583,Z 505.995,A -85,B 0,C 180,E1 19282.972,E2 19282.972} C_VEL
LIN {X 0,Y 417.543,Z 524.549,A -85,B 0,C 180,E1 19282.432,E2 19282.432} C_VEL
LIN {X 0,Y 417.229,Z 542.088,A -85,B 0,C 180,E1 19281.657,E2 19281.657} C_VEL
LIN {X 0,Y 416.732,Z 557.653,A -85,B 0,C 180,E1 19280.725,E2 19280.725} C_VEL
LIN {X 0,Y 416.052,Z 572.227,A -85,B 0,C 180,E1 19279.599,E2 19279.599} C_VEL
LIN {X 0,Y 415.175,Z 586.885,A -85,B 0,C 180,E1 19278.172,E2 19278.172} C_VEL
LIN {X 0,Y 414.275,Z 599.605,A -85,B 0,C 180,E1 19276.63,E2 19276.63} C_VEL
LIN {X 0,Y 413.375,Z 610.472,A -85,B 0,C 180,E1 19274.999,E2 19274.999} C_VEL
LIN {X 0,Y 412.487,Z 620.348,A -85,B 0,C 180,E1 19273.17,E2 19273.17} C_VEL
LIN {X 0,Y 411.666,Z 629.172,A -85,B 0,C 180,E1 19271.114,E2 19271.114} C_VEL
LIN {X 0,Y 410.985,Z 636.273,A -85,B 0,C 180,E1 19268.957,E2 19268.957} C_VEL
LIN {X 0,Y 410.43,Z 641.624,A -85,B 0,C 180,E1 19266.715,E2 19266.715} C_VEL
LIN {X 0,Y 410.031,Z 645.358,A -85,B 0,C 180,E1 19264.335,E2 19264.335} C_VEL
LIN {X 0,Y 409.796,Z 647.151,A -85,B 0,C 180,E1 19262.097,E2 19262.097} C_VEL
LIN {X 0,Y 409.649,Z 647.24,A -85,B 0,C 180,E1 19259.72,E2 19259.72} C_VEL
LIN {X 0,Y 409.605,Z 645.566,A -85,B 0,C 180,E1 19257.341,E2 19257.341} C_VEL
LIN {X 0,Y 409.693,Z 642.114,A -85,B 0,C 180,E1 19254.959,E2 19254.959} C_VEL
LIN {X 0,Y 409.905,Z 637.059,A -85,B 0,C 180,E1 19252.712,E2 19252.712} C_VEL
LIN {X 0,Y 410.292,Z 630.163,A -85,B 0,C 180,E1 19250.461,E2 19250.461} C_VEL
LIN {X 0,Y 410.822,Z 621.81,A -85,B 0,C 180,E1 19248.345,E2 19248.345} C_VEL
LIN {X 0,Y 411.499,Z 611.978,A -85,B 0,C 180,E1 19246.367,E2 19246.367} C_VEL
LIN {X 0,Y 412.377,Z 599.77,A -85,B 0,C 180,E1 19244.387,E2 19244.387} C_VEL
LIN {X 0,Y 413.286,Z 586.892,A -85,B 0,C 180,E1 19242.688,E2 19242.688} C_VEL
LIN {X 0,Y 414.238,Z 572.136,A -85,B 0,C 180,E1 19241.118,E2 19241.118} C_VEL
LIN {X 0,Y 415.138,Z 556.497,A -85,B 0,C 180,E1 19239.78,E2 19239.78} C_VEL
LIN {X 0,Y 415.878,Z 540.66,A -85,B 0,C 180,E1 19238.713,E2 19238.713} C_VEL
LIN {X 0,Y 416.488,Z 522.789,A -85,B 0,C 180,E1 19237.806,E2 19237.806} C_VEL
LIN {X 0,Y 416.891,Z 504.636,A -85,B 0,C 180,E1 19237.159,E2 19237.159} C_VEL
LIN {X 0,Y 417.395,Z 466.689,A -85,B 0,C 180,E1 19236.375,E2 19236.375} C_VEL
LIN {X 0,Y 420.33,Z 337.047,A -85,B 0,C 180,E1 19233.769,E2 19233.769} C_VEL
LIN {X 0,Y 419.88,Z 333.752,A -85,B 0,C 180,E1 19233.652,E2 19233.652} C_VEL
LIN {X 0,Y 420.839,Z 334.53,A -85,B 0,C 180,E1 19233.47,E2 19233.47} C_VEL
LIN {X 0,Y 422.561,Z 333.93,A -85,B 0,C 180,E1 19233.207,E2 19233.207} C_VEL
LIN {X 0,Y 426.135,Z 330.998,A -85,B 0,C 180,E1 19232.73,E2 19232.73} C_VEL
LIN {X 0,Y 428.329,Z 328.287,A -85,B 0,C 180,E1 19232.471,E2 19232.471} C_VEL
LIN {X 0,Y 431.848,Z 327.373,A -85,B 0,C 180,E1 19231.965,E2 19231.965} C_VEL
LIN {X 0,Y 436.059,Z 324.269,A -85,B 0,C 180,E1 19231.44,E2 19231.44} C_VEL
LIN {X 0,Y 438.035,Z 322.516,A -85,B 0,C 180,E1 19231.208,E2 19231.208} C_VEL
LIN {X 0,Y 442.707,Z 320.484,A -85,B 0,C 180,E1 19230.615,E2 19230.615} C_VEL
LIN {X 0,Y 446.264,Z 317.895,A -85,B 0,C 180,E1 19230.211,E2 19230.211} C_VEL
LIN {X 0,Y 438.873,Z 481.851,A -85,B 0,C 180,E1 19226.869,E2 19226.869} C_VEL
LIN {X 0,Y 437.625,Z 502.927,A -85,B 0,C 180,E1 19226.204,E2 19226.204} C_VEL
LIN {X 0,Y 435.863,Z 523.4,A -85,B 0,C 180,E1 19225.325,E2 19225.325} C_VEL
LIN {X 0,Y 433.695,Z 543.099,A -85,B 0,C 180,E1 19224.245,E2 19224.245} C_VEL
LIN {X 0,Y 431.864,Z 556.99,A -85,B 0,C 180,E1 19223.314,E2 19223.314} C_VEL
LIN {X 0,Y 430.06,Z 563.947,A -85,B 0,C 180,E1 19222.887,E2 19222.887} C_VEL
LIN {X 0,Y 422.516,Z 581.115,A -85,B 0,C 180,E1 19221.949,E2 19221.949} C_VEL
LIN {X 0,Y 420.574,Z 587.529,A -85,B 0,C 180,E1 19221.422,E2 19221.422} C_VEL
LIN {X 0,Y 417.272,Z 605.329,A -85,B 0,C 180,E1 19219.506,E2 19219.506} C_VEL
LIN {X 0,Y 414.091,Z 621.532,A -85,B 0,C 180,E1 19217.43,E2 19217.43} C_VEL
LIN {X 0,Y 410.957,Z 637.105,A -85,B 0,C 180,E1 19215.073,E2 19215.073} C_VEL
LIN {X 0,Y 408.124,Z 651.218,A -85,B 0,C 180,E1 19212.545,E2 19212.545} C_VEL
LIN {X 0,Y 405.696,Z 663.919,A -85,B 0,C 180,E1 19209.851,E2 19209.851} C_VEL
LIN {X 0,Y 403.7,Z 675.054,A -85,B 0,C 180,E1 19207.003,E2 19207.003} C_VEL
LIN {X 0,Y 402.215,Z 684.393,A -85,B 0,C 180,E1 19204.126,E2 19204.126} C_VEL
LIN {X 0,Y 401.111,Z 692.721,A -85,B 0,C 180,E1 19200.962,E2 19200.962} C_VEL
LIN {X 0,Y 400.495,Z 699.048,A -85,B 0,C 180,E1 19197.897,E2 19197.897} C_VEL
LIN {X 0,Y 400.166,Z 703.683,A -85,B 0,C 180,E1 19194.82,E2 19194.82} C_VEL
LIN {X 0,Y 400.034,Z 706.801,A -85,B 0,C 180,E1 19191.711,E2 19191.711} C_VEL
LIN {X 0,Y 399.989,Z 708.396,A -85,B 0,C 180,E1 19188.661,E2 19188.661} C_VEL
LIN {X 0,Y 399.995,Z 708.464,A -85,B 0,C 180,E1 19185.764,E2 19185.764} C_VEL
LIN {X 0,Y 400.013,Z 707.149,A -85,B 0,C 180,E1 19182.707,E2 19182.707} C_VEL
LIN {X 0,Y 400.127,Z 704.337,A -85,B 0,C 180,E1 19179.638,E2 19179.638} C_VEL
LIN {X 0,Y 400.392,Z 699.933,A -85,B 0,C 180,E1 19176.596,E2 19176.596} C_VEL
LIN {X 0,Y 400.979,Z 693.722,A -85,B 0,C 180,E1 19173.431,E2 19173.431} C_VEL
LIN {X 0,Y 401.925,Z 686.177,A -85,B 0,C 180,E1 19170.428,E2 19170.428} C_VEL
LIN {X 0,Y 403.349,Z 676.798,A -85,B 0,C 180,E1 19167.443,E2 19167.443} C_VEL
LIN {X 0,Y 405.214,Z 666.05,A -85,B 0,C 180,E1 19164.62,E2 19164.62} C_VEL
LIN {X 0,Y 407.625,Z 653.289,A -85,B 0,C 180,E1 19161.821,E2 19161.821} C_VEL
LIN {X 0,Y 410.322,Z 639.815,A -85,B 0,C 180,E1 19159.328,E2 19159.328} C_VEL
LIN {X 0,Y 413.293,Z 624.92,A -85,B 0,C 180,E1 19156.998,E2 19156.998} C_VEL
LIN {X 0,Y 416.38,Z 608.966,A -85,B 0,C 180,E1 19154.898,E2 19154.898} C_VEL
LIN {X 0,Y 419.588,Z 591.563,A -85,B 0,C 180,E1 19152.956,E2 19152.956} C_VEL
LIN {X 0,Y 422.624,Z 573.955,A -85,B 0,C 180,E1 19151.303,E2 19151.303} C_VEL
LIN {X 0,Y 425.442,Z 555.454,A -85,B 0,C 180,E1 19149.861,E2 19149.861} C_VEL
LIN {X 0,Y 427.937,Z 536.051,A -85,B 0,C 180,E1 19148.624,E2 19148.624} C_VEL
LIN {X 0,Y 430.176,Z 515.044,A -85,B 0,C 180,E1 19147.557,E2 19147.557} C_VEL
LIN {X 0,Y 431.867,Z 494.561,A -85,B 0,C 180,E1 19146.762,E2 19146.762} C_VEL
LIN {X 0,Y 432.968,Z 474.042,A -85,B 0,C 180,E1 19146.195,E2 19146.195} C_VEL
LIN {X 0,Y 441.015,Z 296.391,A -85,B 0,C 180,E1 19142.607,E2 19142.607} C_VEL
LIN {X 0,Y 442.783,Z 251.204,A -85,B 0,C 180,E1 19141.724,E2 19141.724} C_VEL
LIN {X 0,Y 434.038,Z 238.328,A -85,B 0,C 180,E1 19140.282,E2 19140.282} C_VEL
LIN {X 0,Y 420.245,Z 221.847,A -85,B 0,C 180,E1 19137.946,E2 19137.946} C_VEL
LIN {X 0,Y 413.836,Z 214.563,A -85,B 0,C 180,E1 19136.78,E2 19136.78} C_VEL
LIN {X 0,Y 411.966,Z 210.996,A -85,B 0,C 180,E1 19135.856,E2 19135.856} C_VEL
LIN {X 0,Y 409.521,Z 206.478,A -85,B 0,C 180,E1 19134.635,E2 19134.635} C_VEL
LIN {X 0,Y 406.81,Z 201.648,A -85,B 0,C 180,E1 19133.25,E2 19133.25} C_VEL
LIN {X 0,Y 404.684,Z 197.922,A -85,B 0,C 180,E1 19132.13,E2 19132.13} C_VEL
LIN {X 0,Y 404.113,Z 196.734,A -85,B 0,C 180,E1 19131.79,E2 19131.79} C_VEL
LIN {X 0,Y 401.93,Z 193.509,A -85,B 0,C 180,E1 19130.684,E2 19130.684} C_VEL
LIN {X 0,Y 401.468,Z 191.728,A -85,B 0,C 180,E1 19130.204,E2 19130.204} C_VEL
LIN {X 0,Y 401.489,Z 191.724,A -85,B 0,C 180,E1 19126.238,E2 19126.238} C_VEL
LIN {X 0,Y 401.504,Z 191.719,A -85,B 0,C 180,E1 19122.251,E2 19122.251} C_VEL
LIN {X 0,Y 401.501,Z 191.722,A -85,B 0,C 180,E1 19118.323,E2 19118.323} C_VEL
LIN {X 0,Y 401.474,Z 191.727,A -85,B 0,C 180,E1 19114.426,E2 19114.426} C_VEL
LIN {X 0,Y 401.486,Z 191.717,A -85,B 0,C 180,E1 19110.495,E2 19110.495} C_VEL
LIN {X 0,Y 401.499,Z 191.705,A -85,B 0,C 180,E1 19106.617,E2 19106.617} C_VEL
LIN {X 0,Y 401.504,Z 191.697,A -85,B 0,C 180,E1 19102.706,E2 19102.706} C_VEL
LIN {X 0,Y 401.491,Z 191.704,A -85,B 0,C 180,E1 19098.74,E2 19098.74} C_VEL
LIN {X 0,Y 401.47,Z 191.719,A -85,B 0,C 180,E1 19094.864,E2 19094.864} C_VEL
LIN {X 0,Y 401.479,Z 191.728,A -85,B 0,C 180,E1 19090.911,E2 19090.911} C_VEL
LIN {X 0,Y 401.509,Z 191.717,A -85,B 0,C 180,E1 19087.009,E2 19087.009} C_VEL
LIN {X 0,Y 401.496,Z 191.711,A -85,B 0,C 180,E1 19082.998,E2 19082.998} C_VEL
LIN {X 0,Y 401.479,Z 191.71,A -85,B 0,C 180,E1 19079.002,E2 19079.002} C_VEL
LIN {X 0,Y 401.455,Z 191.711,A -85,B 0,C 180,E1 19075.143,E2 19075.143} C_VEL
LIN {X 0,Y 401.443,Z 191.713,A -85,B 0,C 180,E1 19071.262,E2 19071.262} C_VEL
LIN {X 0,Y 401.48,Z 191.802,A -85,B 0,C 180,E1 19067.707,E2 19067.707} C_VEL
LIN {X 0,Y 402.803,Z 195.196,A -85,B 0,C 180,E1 19066.8,E2 19066.8} C_VEL
LIN {X 0,Y 404.562,Z 197.495,A -85,B 0,C 180,E1 19065.984,E2 19065.984} C_VEL
LIN {X 0,Y 406.576,Z 201.315,A -85,B 0,C 180,E1 19064.89,E2 19064.89} C_VEL
LIN {X 0,Y 407.434,Z 202.623,A -85,B 0,C 180,E1 19064.485,E2 19064.485} C_VEL
LIN {X 0,Y 409.58,Z 206.54,A -85,B 0,C 180,E1 19063.405,E2 19063.405} C_VEL
LIN {X 0,Y 413.445,Z 213.825,A -85,B 0,C 180,E1 19061.531,E2 19061.531} C_VEL
LIN {X 0,Y 418.09,Z 222.513,A -85,B 0,C 180,E1 19059.418,E2 19059.418} C_VEL
LIN {X 0,Y 424.355,Z 234.984,A -85,B 0,C 180,E1 19056.682,E2 19056.682} C_VEL
LIN {X 0,Y 431.47,Z 249.916,A -85,B 0,C 180,E1 19053.73,E2 19053.73} C_VEL
LIN {X 0,Y 439.721,Z 268.644,A -85,B 0,C 180,E1 19050.434,E2 19050.434} C_VEL
LIN {X 0,Y 440.111,Z 270.255,A -85,B 0,C 180,E1 19050.208,E2 19050.208} C_VEL
LIN {X 0,Y 434.594,Z 322.142,A -85,B 0,C 180,E1 19045.531,E2 19045.531} C_VEL
LIN {X 0,Y 434.735,Z 341.308,A -85,B 0,C 180,E1 19043.603,E2 19043.603} C_VEL
LIN {X 0,Y 436.75,Z 358.135,A -85,B 0,C 180,E1 19041.742,E2 19041.742} C_VEL
LIN {X 0,Y 440.748,Z 374.22,A -85,B 0,C 180,E1 19039.805,E2 19039.805} C_VEL
LIN {X 0,Y 446.411,Z 388.34,A -85,B 0,C 180,E1 19037.957,E2 19037.957} C_VEL
LIN {X 0,Y 453.57,Z 400.779,A -85,B 0,C 180,E1 19036.197,E2 19036.197} C_VEL
LIN {X 0,Y 462.984,Z 412.636,A -85,B 0,C 180,E1 19034.371,E2 19034.371} C_VEL
LIN {X 0,Y 465.137,Z 415.282,A -85,B 0,C 180,E1 19033.973,E2 19033.973} C_VEL
LIN {X 0,Y 455.776,Z 431.412,A -85,B 0,C 180,E1 19033.365,E2 19033.365} C_VEL
LIN {X 0,Y 446.396,Z 447.506,A -85,B 0,C 180,E1 19032.74,E2 19032.74} C_VEL
LIN {X 0,Y 440.827,Z 459.25,A -85,B 0,C 180,E1 19032.208,E2 19032.208} C_VEL
LIN {X 0,Y 437.575,Z 481.412,A -85,B 0,C 180,E1 19032.1,E2 19032.1} C_VEL
LIN {X 0,Y 436.073,Z 499.079,A -85,B 0,C 180,E1 19031.864,E2 19031.864} C_VEL
LIN {X 0,Y 434.167,Z 525.219,A -85,B 0,C 180,E1 19031.217,E2 19031.217} C_VEL
LIN {X 0,Y 431.352,Z 550.634,A -85,B 0,C 180,E1 19030.376,E2 19030.376} C_VEL
LIN {X 0,Y 428.374,Z 574.378,A -85,B 0,C 180,E1 19029.324,E2 19029.324} C_VEL
LIN {X 0,Y 425.165,Z 597.286,A -85,B 0,C 180,E1 19028.035,E2 19028.035} C_VEL
LIN {X 0,Y 421.864,Z 619.441,A -85,B 0,C 180,E1 19026.505,E2 19026.505} C_VEL
LIN {X 0,Y 418.482,Z 640.742,A -85,B 0,C 180,E1 19024.725,E2 19024.725} C_VEL
LIN {X 0,Y 415.318,Z 660.16,A -85,B 0,C 180,E1 19022.798,E2 19022.798} C_VEL
LIN {X 0,Y 412.075,Z 679.274,A -85,B 0,C 180,E1 19020.53,E2 19020.53} C_VEL
LIN {X 0,Y 409.278,Z 695.711,A -85,B 0,C 180,E1 19018.211,E2 19018.211} C_VEL
LIN {X 0,Y 406.849,Z 710.466,A -85,B 0,C 180,E1 19015.784,E2 19015.784} C_VEL
LIN {X 0,Y 404.601,Z 724.822,A -85,B 0,C 180,E1 19012.983,E2 19012.983} C_VEL
LIN {X 0,Y 402.962,Z 736.429,A -85,B 0,C 180,E1 19010.296,E2 19010.296} C_VEL
LIN {X 0,Y 401.666,Z 747.017,A -85,B 0,C 180,E1 19007.38,E2 19007.38} C_VEL
LIN {X 0,Y 400.784,Z 756.094,A -85,B 0,C 180,E1 19004.299,E2 19004.299} C_VEL
LIN {X 0,Y 400.298,Z 762.934,A -85,B 0,C 180,E1 19001.38,E2 19001.38} C_VEL
LIN {X 0,Y 400.057,Z 768.525,A -85,B 0,C 180,E1 18998.226,E2 18998.226} C_VEL
LIN {X 0,Y 399.99,Z 772.154,A -85,B 0,C 180,E1 18995.163,E2 18995.163} C_VEL
LIN {X 0,Y 399.983,Z 774.071,A -85,B 0,C 180,E1 18992.292,E2 18992.292} C_VEL
LIN {X 0,Y 399.981,Z 774.45,A -85,B 0,C 180,E1 18989.284,E2 18989.284} C_VEL
LIN {X 0,Y 399.981,Z 773.346,A -85,B 0,C 180,E1 18986.417,E2 18986.417} C_VEL
LIN {X 0,Y 400.007,Z 770.545,A -85,B 0,C 180,E1 18983.397,E2 18983.397} C_VEL
LIN {X 0,Y 400.134,Z 766.335,A -85,B 0,C 180,E1 18980.507,E2 18980.507} C_VEL
LIN {X 0,Y 400.483,Z 759.809,A -85,B 0,C 180,E1 18977.308,E2 18977.308} C_VEL
LIN {X 0,Y 401.15,Z 751.622,A -85,B 0,C 180,E1 18974.235,E2 18974.235} C_VEL
LIN {X 0,Y 402.173,Z 741.888,A -85,B 0,C 180,E1 18971.294,E2 18971.294} C_VEL
LIN {X 0,Y 403.684,Z 730.026,A -85,B 0,C 180,E1 18968.343,E2 18968.343} C_VEL
LIN {X 0,Y 405.626,Z 716.491,A -85,B 0,C 180,E1 18965.536,E2 18965.536} C_VEL
LIN {X 0,Y 407.842,Z 702.225,A -85,B 0,C 180,E1 18963.028,E2 18963.028} C_VEL
LIN {X 0,Y 410.549,Z 685.517,A -85,B 0,C 180,E1 18960.53,E2 18960.53} C_VEL
LIN {X 0,Y 413.464,Z 667.602,A -85,B 0,C 180,E1 18958.266,E2 18958.266} C_VEL
LIN {X 0,Y 416.553,Z 648.692,A -85,B 0,C 180,E1 18956.243,E2 18956.243} C_VEL
LIN {X 0,Y 419.615,Z 628.77,A -85,B 0,C 180,E1 18954.45,E2 18954.45} C_VEL
LIN {X 0,Y 423.016,Z 606.568,A -85,B 0,C 180,E1 18952.764,E2 18952.764} C_VEL
LIN {X 0,Y 426.153,Z 584.502,A -85,B 0,C 180,E1 18951.383,E2 18951.383} C_VEL
LIN {X 0,Y 429.372,Z 560.536,A -85,B 0,C 180,E1 18950.179,E2 18950.179} C_VEL
LIN {X 0,Y 432.297,Z 537.059,A -85,B 0,C 180,E1 18949.249,E2 18949.249} C_VEL
LIN {X 0,Y 434.916,Z 510.639,A -85,B 0,C 180,E1 18948.468,E2 18948.468} C_VEL
LIN {X 0,Y 436.506,Z 488.028,A -85,B 0,C 180,E1 18947.982,E2 18947.982} C_VEL
LIN {X 0,Y 438.72,Z 464.385,A -85,B 0,C 180,E1 18947.726,E2 18947.726} C_VEL
LIN {X 0,Y 440.51,Z 447.414,A -85,B 0,C 180,E1 18947.569,E2 18947.569} C_VEL
LIN {X 0,Y 447.637,Z 427.083,A -85,B 0,C 180,E1 18946.919,E2 18946.919} C_VEL
LIN {X 0,Y 456.404,Z 401.488,A -85,B 0,C 180,E1 18946.102,E2 18946.102} C_VEL
LIN {X 0,Y 466.107,Z 378.127,A -85,B 0,C 180,E1 18945.542,E2 18945.542} C_VEL
LIN {X 0,Y 480.328,Z 348.301,A -85,B 0,C 180,E1 18945.023,E2 18945.023} C_VEL
LIN {X 0,Y 485.297,Z 338.166,A -85,B 0,C 180,E1 18944.867,E2 18944.867} C_VEL
LIN {X 0,Y 486.413,Z 334.499,A -85,B 0,C 180,E1 18944.747,E2 18944.747} C_VEL
LIN {X 0,Y 475.735,Z 324.9,A -85,B 0,C 180,E1 18943.083,E2 18943.083} C_VEL
LIN {X 0,Y 465.995,Z 312.866,A -85,B 0,C 180,E1 18941.201,E2 18941.201} C_VEL
LIN {X 0,Y 459.058,Z 300.767,A -85,B 0,C 180,E1 18939.493,E2 18939.493} C_VEL
LIN {X 0,Y 448.033,Z 273.173,A -85,B 0,C 180,E1 18935.811,E2 18935.811} C_VEL
LIN {X 0,Y 438.388,Z 278.978,A -85,B 0,C 180,E1 18934.763,E2 18934.763} C_VEL
LIN {X 0,Y 433.388,Z 281.845,A -85,B 0,C 180,E1 18934.178,E2 18934.178} C_VEL
LIN {X 0,Y 428.938,Z 285.009,A -85,B 0,C 180,E1 18933.695,E2 18933.695} C_VEL
LIN {X 0,Y 426.336,Z 286.333,A -85,B 0,C 180,E1 18933.356,E2 18933.356} C_VEL
LIN {X 0,Y 422.706,Z 289.199,A -85,B 0,C 180,E1 18932.958,E2 18932.958} C_VEL
LIN {X 0,Y 420.065,Z 290.048,A -85,B 0,C 180,E1 18932.543,E2 18932.543} C_VEL
LIN {X 0,Y 418.758,Z 329.38,A -85,B 0,C 180,E1 18928.992,E2 18928.992} C_VEL
LIN {X 0,Y 418.077,Z 344.348,A -85,B 0,C 180,E1 18927.643,E2 18927.643} C_VEL
LIN {X 0,Y 415.843,Z 353.795,A -85,B 0,C 180,E1 18927.047,E2 18927.047} C_VEL
LIN {X 0,Y 411.521,Z 454.649,A -85,B 0,C 180,E1 18924.601,E2 18924.601} C_VEL
LIN {X 0,Y 410.312,Z 507.789,A -85,B 0,C 180,E1 18923.399,E2 18923.399} C_VEL
LIN {X 0,Y 410.267,Z 526.439,A -85,B 0,C 180,E1 18922.842,E2 18922.842} C_VEL
LIN {X 0,Y 409.915,Z 543.97,A -85,B 0,C 180,E1 18922.044,E2 18922.044} C_VEL
LIN {X 0,Y 409.344,Z 560.204,A -85,B 0,C 180,E1 18921.042,E2 18921.042} C_VEL
LIN {X 0,Y 408.562,Z 575.522,A -85,B 0,C 180,E1 18919.812,E2 18919.812} C_VEL
LIN {X 0,Y 407.687,Z 589.112,A -85,B 0,C 180,E1 18918.443,E2 18918.443} C_VEL
LIN {X 0,Y 406.716,Z 601.781,A -85,B 0,C 180,E1 18916.863,E2 18916.863} C_VEL
LIN {X 0,Y 405.728,Z 612.903,A -85,B 0,C 180,E1 18915.142,E2 18915.142} C_VEL
LIN {X 0,Y 404.724,Z 623.285,A -85,B 0,C 180,E1 18913.137,E2 18913.137} C_VEL
LIN {X 0,Y 403.9,Z 631.486,A -85,B 0,C 180,E1 18911.133,E2 18911.133} C_VEL
LIN {X 0,Y 403.187,Z 638.216,A -85,B 0,C 180,E1 18908.988,E2 18908.988} C_VEL
LIN {X 0,Y 402.598,Z 643.428,A -85,B 0,C 180,E1 18906.703,E2 18906.703} C_VEL
LIN {X 0,Y 402.19,Z 646.84,A -85,B 0,C 180,E1 18904.42,E2 18904.42} C_VEL
LIN {X 0,Y 401.929,Z 648.582,A -85,B 0,C 180,E1 18902.138,E2 18902.138} C_VEL
LIN {X 0,Y 401.767,Z 648.609,A -85,B 0,C 180,E1 18899.714,E2 18899.714} C_VEL
LIN {X 0,Y 401.717,Z 646.857,A -85,B 0,C 180,E1 18897.289,E2 18897.289} C_VEL
LIN {X 0,Y 401.797,Z 643.559,A -85,B 0,C 180,E1 18895.003,E2 18895.003} C_VEL
LIN {X 0,Y 402.012,Z 638.517,A -85,B 0,C 180,E1 18892.712,E2 18892.712} C_VEL
LIN {X 0,Y 402.412,Z 631.62,A -85,B 0,C 180,E1 18890.417,E2 18890.417} C_VEL
LIN {X 0,Y 402.96,Z 623.259,A -85,B 0,C 180,E1 18888.26,E2 18888.26} C_VEL
LIN {X 0,Y 403.664,Z 613.43,A -85,B 0,C 180,E1 18886.243,E2 18886.243} C_VEL
LIN {X 0,Y 404.574,Z 601.218,A -85,B 0,C 180,E1 18884.225,E2 18884.225} C_VEL
LIN {X 0,Y 405.518,Z 588.341,A -85,B 0,C 180,E1 18882.493,E2 18882.493} C_VEL
LIN {X 0,Y 406.5,Z 573.7,A -85,B 0,C 180,E1 18880.904,E2 18880.904} C_VEL
LIN {X 0,Y 407.441,Z 557.986,A -85,B 0,C 180,E1 18879.531,E2 18879.531} C_VEL
LIN {X 0,Y 408.216,Z 542.249,A -85,B 0,C 180,E1 18878.444,E2 18878.444} C_VEL
LIN {X 0,Y 408.854,Z 524.413,A -85,B 0,C 180,E1 18877.516,E2 18877.516} C_VEL
LIN {X 0,Y 409.286,Z 506.14,A -85,B 0,C 180,E1 18876.844,E2 18876.844} C_VEL
LIN {X 0,Y 409.738,Z 472.296,A -85,B 0,C 180,E1 18876.115,E2 18876.115} C_VEL
LIN {X 0,Y 412.47,Z 364.575,A -85,B 0,C 180,E1 18873.897,E2 18873.897} C_VEL
LIN {X 0,Y 413.271,Z 365.855,A -85,B 0,C 180,E1 18873.72,E2 18873.72} C_VEL
LIN {X 0,Y 414.478,Z 365.54,A -85,B 0,C 180,E1 18873.53,E2 18873.53} C_VEL
LIN {X 0,Y 416.657,Z 362.212,A -85,B 0,C 180,E1 18873.278,E2 18873.278} C_VEL
LIN {X 0,Y 420.076,Z 353.298,A -85,B 0,C 180,E1 18873.007,E2 18873.007} C_VEL
LIN {X 0,Y 423.559,Z 341.406,A -85,B 0,C 180,E1 18872.82,E2 18872.82} C_VEL
LIN {X 0,Y 428.128,Z 337.837,A -85,B 0,C 180,E1 18872.222,E2 18872.222} C_VEL
LIN {X 0,Y 430.056,Z 335.862,A -85,B 0,C 180,E1 18871.989,E2 18871.989} C_VEL
LIN {X 0,Y 434.661,Z 333.817,A -85,B 0,C 180,E1 18871.377,E2 18871.377} C_VEL
LIN {X 0,Y 439.554,Z 329.936,A -85,B 0,C 180,E1 18870.795,E2 18870.795} C_VEL
LIN {X 0,Y 440.129,Z 329.942,A -85,B 0,C 180,E1 18870.716,E2 18870.716} C_VEL
LIN {X 0,Y 432.651,Z 483.055,A -85,B 0,C 180,E1 18867.514,E2 18867.514} C_VEL
LIN {X 0,Y 431.339,Z 504.459,A -85,B 0,C 180,E1 18866.829,E2 18866.829} C_VEL
LIN {X 0,Y 429.551,Z 524.451,A -85,B 0,C 180,E1 18865.961,E2 18865.961} C_VEL
LIN {X 0,Y 427.338,Z 543.473,A -85,B 0,C 180,E1 18864.903,E2 18864.903} C_VEL
LIN {X 0,Y 424.694,Z 562.193,A -85,B 0,C 180,E1 18863.609,E2 18863.609} C_VEL
LIN {X 0,Y 421.529,Z 581.885,A -85,B 0,C 180,E1 18861.953,E2 18861.953} C_VEL
LIN {X 0,Y 420.574,Z 587.529,A -85,B 0,C 180,E1 18861.422,E2 18861.422} C_VEL
LIN {X 0,Y 418.581,Z 593.859,A -85,B 0,C 180,E1 18860.861,E2 18860.861} C_VEL
LIN {X 0,Y 410.521,Z 609.811,A -85,B 0,C 180,E1 18859.566,E2 18859.566} C_VEL
LIN {X 0,Y 408.523,Z 615.551,A -85,B 0,C 180,E1 18858.916,E2 18858.916} C_VEL
LIN {X 0,Y 405.234,Z 631.081,A -85,B 0,C 180,E1 18856.691,E2 18856.691} C_VEL
LIN {X 0,Y 402.008,Z 646.14,A -85,B 0,C 180,E1 18854.14,E2 18854.14} C_VEL
LIN {X 0,Y 399.276,Z 659.19,A -85,B 0,C 180,E1 18851.517,E2 18851.517} C_VEL
LIN {X 0,Y 396.915,Z 671.162,A -85,B 0,C 180,E1 18848.655,E2 18848.655} C_VEL
LIN {X 0,Y 395.018,Z 681.663,A -85,B 0,C 180,E1 18845.604,E2 18845.604} C_VEL
LIN {X 0,Y 393.677,Z 690.307,A -85,B 0,C 180,E1 18842.518,E2 18842.518} C_VEL
LIN {X 0,Y 392.779,Z 697.551,A -85,B 0,C 180,E1 18839.259,E2 18839.259} C_VEL
LIN {X 0,Y 392.326,Z 702.792,A -85,B 0,C 180,E1 18836.161,E2 18836.161} C_VEL
LIN {X 0,Y 392.105,Z 706.359,A -85,B 0,C 180,E1 18833.123,E2 18833.123} C_VEL
LIN {X 0,Y 392.033,Z 708.547,A -85,B 0,C 180,E1 18829.984,E2 18829.984} C_VEL
LIN {X 0,Y 392.018,Z 709.298,A -85,B 0,C 180,E1 18826.904,E2 18826.904} C_VEL
LIN {X 0,Y 392.041,Z 708.495,A -85,B 0,C 180,E1 18823.871,E2 18823.871} C_VEL
LIN {X 0,Y 392.099,Z 706.244,A -85,B 0,C 180,E1 18820.729,E2 18820.729} C_VEL
LIN {X 0,Y 392.334,Z 702.535,A -85,B 0,C 180,E1 18817.616,E2 18817.616} C_VEL
LIN {X 0,Y 392.787,Z 697.202,A -85,B 0,C 180,E1 18814.526,E2 18814.526} C_VEL
LIN {X 0,Y 393.687,Z 689.958,A -85,B 0,C 180,E1 18811.31,E2 18811.31} C_VEL
LIN {X 0,Y 395.009,Z 681.344,A -85,B 0,C 180,E1 18808.26,E2 18808.26} C_VEL
LIN {X 0,Y 396.892,Z 670.847,A -85,B 0,C 180,E1 18805.231,E2 18805.231} C_VEL
LIN {X 0,Y 399.236,Z 658.801,A -85,B 0,C 180,E1 18802.373,E2 18802.373} C_VEL
LIN {X 0,Y 401.86,Z 646.04,A -85,B 0,C 180,E1 18799.825,E2 18799.825} C_VEL
LIN {X 0,Y 404.817,Z 632.046,A -85,B 0,C 180,E1 18797.447,E2 18797.447} C_VEL
LIN {X 0,Y 408.057,Z 616.48,A -85,B 0,C 180,E1 18795.2,E2 18795.2} C_VEL
LIN {X 0,Y 411.339,Z 599.801,A -85,B 0,C 180,E1 18793.187,E2 18793.187} C_VEL
LIN {X 0,Y 414.499,Z 582.63,A -85,B 0,C 180,E1 18791.433,E2 18791.433} C_VEL
LIN {X 0,Y 417.493,Z 564.847,A -85,B 0,C 180,E1 18789.9,E2 18789.9} C_VEL
LIN {X 0,Y 420.369,Z 545.289,A -85,B 0,C 180,E1 18788.513,E2 18788.513} C_VEL
LIN {X 0,Y 422.595,Z 526.879,A -85,B 0,C 180,E1 18787.462,E2 18787.462} C_VEL
LIN {X 0,Y 424.641,Z 506.02,A -85,B 0,C 180,E1 18786.519,E2 18786.519} C_VEL
LIN {X 0,Y 426.095,Z 485.361,A -85,B 0,C 180,E1 18785.819,E2 18785.819} C_VEL
LIN {X 0,Y 428.824,Z 427.847,A -85,B 0,C 180,E1 18784.562,E2 18784.562} C_VEL
LIN {X 0,Y 435.472,Z 290.533,A -85,B 0,C 180,E1 18781.768,E2 18781.768} C_VEL
LIN {X 0,Y 436.97,Z 254.862,A -85,B 0,C 180,E1 18781.072,E2 18781.072} C_VEL
LIN {X 0,Y 429.518,Z 244.025,A -85,B 0,C 180,E1 18779.813,E2 18779.813} C_VEL
LIN {X 0,Y 416.133,Z 227.933,A -85,B 0,C 180,E1 18777.498,E2 18777.498} C_VEL
LIN {X 0,Y 407.557,Z 217.855,A -85,B 0,C 180,E1 18775.894,E2 18775.894} C_VEL
LIN {X 0,Y 403.793,Z 211.472,A -85,B 0,C 180,E1 18774.066,E2 18774.066} C_VEL
LIN {X 0,Y 401.743,Z 207.633,A -85,B 0,C 180,E1 18772.966,E2 18772.966} C_VEL
LIN {X 0,Y 398.942,Z 202.671,A -85,B 0,C 180,E1 18771.441,E2 18771.441} C_VEL
LIN {X 0,Y 396.791,Z 198.795,A -85,B 0,C 180,E1 18770.205,E2 18770.205} C_VEL
LIN {X 0,Y 396.233,Z 197.775,A -85,B 0,C 180,E1 18769.872,E2 18769.872} C_VEL
LIN {X 0,Y 394.047,Z 194.623,A -85,B 0,C 180,E1 18768.684,E2 18768.684} C_VEL
LIN {X 0,Y 393.536,Z 192.695,A -85,B 0,C 180,E1 18768.111,E2 18768.111} C_VEL
LIN {X 0,Y 393.555,Z 192.692,A -85,B 0,C 180,E1 18764.117,E2 18764.117} C_VEL
LIN {X 0,Y 393.561,Z 192.69,A -85,B 0,C 180,E1 18760.12,E2 18760.12} C_VEL
LIN {X 0,Y 393.539,Z 192.691,A -85,B 0,C 180,E1 18756.298,E2 18756.298} C_VEL
LIN {X 0,Y 393.529,Z 192.692,A -85,B 0,C 180,E1 18752.419,E2 18752.419} C_VEL
LIN {X 0,Y 393.555,Z 192.698,A -85,B 0,C 180,E1 18748.531,E2 18748.531} C_VEL
LIN {X 0,Y 393.562,Z 192.71,A -85,B 0,C 180,E1 18744.562,E2 18744.562} C_VEL
LIN {X 0,Y 393.567,Z 192.711,A -85,B 0,C 180,E1 18740.524,E2 18740.524} C_VEL
LIN {X 0,Y 393.558,Z 192.705,A -85,B 0,C 180,E1 18736.532,E2 18736.532} C_VEL
LIN {X 0,Y 393.538,Z 192.693,A -85,B 0,C 180,E1 18732.621,E2 18732.621} C_VEL
LIN {X 0,Y 393.559,Z 192.688,A -85,B 0,C 180,E1 18728.621,E2 18728.621} C_VEL
LIN {X 0,Y 393.561,Z 192.689,A -85,B 0,C 180,E1 18724.664,E2 18724.664} C_VEL
LIN {X 0,Y 393.556,Z 192.696,A -85,B 0,C 180,E1 18720.728,E2 18720.728} C_VEL
LIN {X 0,Y 393.538,Z 192.702,A -85,B 0,C 180,E1 18716.796,E2 18716.796} C_VEL
LIN {X 0,Y 393.518,Z 192.704,A -85,B 0,C 180,E1 18712.849,E2 18712.849} C_VEL
LIN {X 0,Y 393.524,Z 192.755,A -85,B 0,C 180,E1 18709.756,E2 18709.756} C_VEL
LIN {X 0,Y 394.598,Z 195.787,A -85,B 0,C 180,E1 18708.897,E2 18708.897} C_VEL
LIN {X 0,Y 396.604,Z 198.193,A -85,B 0,C 180,E1 18707.922,E2 18707.922} C_VEL
LIN {X 0,Y 398.423,Z 202.018,A -85,B 0,C 180,E1 18706.799,E2 18706.799} C_VEL
LIN {X 0,Y 399.607,Z 203.536,A -85,B 0,C 180,E1 18706.25,E2 18706.25} C_VEL
LIN {X 0,Y 401.587,Z 207.367,A -85,B 0,C 180,E1 18705.141,E2 18705.141} C_VEL
LIN {X 0,Y 405.589,Z 214.676,A -85,B 0,C 180,E1 18703.089,E2 18703.089} C_VEL
LIN {X 0,Y 410.139,Z 222.986,A -85,B 0,C 180,E1 18700.934,E2 18700.934} C_VEL
LIN {X 0,Y 416.523,Z 235.548,A -85,B 0,C 180,E1 18698.008,E2 18698.008} C_VEL
LIN {X 0,Y 423.765,Z 250.705,A -85,B 0,C 180,E1 18694.869,E2 18694.869} C_VEL
LIN {X 0,Y 431.862,Z 268.988,A -85,B 0,C 180,E1 18691.515,E2 18691.515} C_VEL
LIN {X 0,Y 433.855,Z 273.669,A -85,B 0,C 180,E1 18690.712,E2 18690.712} C_VEL
LIN {X 0,Y 428.156,Z 324.567,A -85,B 0,C 180,E1 18686.074,E2 18686.074} C_VEL
LIN {X 0,Y 428.14,Z 343.806,A -85,B 0,C 180,E1 18684.115,E2 18684.115} C_VEL
LIN {X 0,Y 429.957,Z 360.539,A -85,B 0,C 180,E1 18682.248,E2 18682.248} C_VEL
LIN {X 0,Y 433.828,Z 377.073,A -85,B 0,C 180,E1 18680.241,E2 18680.241} C_VEL
LIN {X 0,Y 439.322,Z 391.442,A -85,B 0,C 180,E1 18678.351,E2 18678.351} C_VEL
LIN {X 0,Y 446.819,Z 404.939,A -85,B 0,C 180,E1 18676.432,E2 18676.432} C_VEL
LIN {X 0,Y 456.607,Z 417.514,A -85,B 0,C 180,E1 18674.485,E2 18674.485} C_VEL
LIN {X 0,Y 456.268,Z 418.518,A -85,B 0,C 180,E1 18674.427,E2 18674.427} C_VEL
LIN {X 0,Y 449.772,Z 429.708,A -85,B 0,C 180,E1 18674.003,E2 18674.003} C_VEL
LIN {X 0,Y 439.922,Z 446.602,A -85,B 0,C 180,E1 18673.345,E2 18673.345} C_VEL
LIN {X 0,Y 435.159,Z 456.59,A -85,B 0,C 180,E1 18672.903,E2 18672.903} C_VEL
LIN {X 0,Y 431.57,Z 480.592,A -85,B 0,C 180,E1 18672.794,E2 18672.794} C_VEL
LIN {X 0,Y 429.896,Z 498.855,A -85,B 0,C 180,E1 18672.542,E2 18672.542} C_VEL
LIN {X 0,Y 427.77,Z 525.971,A -85,B 0,C 180,E1 18671.849,E2 18671.849} C_VEL
LIN {X 0,Y 424.844,Z 550.943,A -85,B 0,C 180,E1 18670.998,E2 18670.998} C_VEL
LIN {X 0,Y 421.636,Z 575.071,A -85,B 0,C 180,E1 18669.897,E2 18669.897} C_VEL
LIN {X 0,Y 418.304,Z 597.772,A -85,B 0,C 180,E1 18668.592,E2 18668.592} C_VEL
LIN {X 0,Y 414.876,Z 619.65,A -85,B 0,C 180,E1 18667.049,E2 18667.049} C_VEL
LIN {X 0,Y 411.518,Z 640.001,A -85,B 0,C 180,E1 18665.328,E2 18665.328} C_VEL
LIN {X 0,Y 408.282,Z 658.932,A -85,B 0,C 180,E1 18663.436,E2 18663.436} C_VEL
LIN {X 0,Y 404.794,Z 678.596,A -85,B 0,C 180,E1 18661.08,E2 18661.08} C_VEL
LIN {X 0,Y 401.733,Z 695.724,A -85,B 0,C 180,E1 18658.627,E2 18658.627} C_VEL
LIN {X 0,Y 399.175,Z 710.376,A -85,B 0,C 180,E1 18656.158,E2 18656.158} C_VEL
LIN {X 0,Y 396.817,Z 724.728,A -85,B 0,C 180,E1 18653.303,E2 18653.303} C_VEL
LIN {X 0,Y 394.952,Z 737.308,A -85,B 0,C 180,E1 18650.293,E2 18650.293} C_VEL
LIN {X 0,Y 393.679,Z 747.223,A -85,B 0,C 180,E1 18647.439,E2 18647.439} C_VEL
LIN {X 0,Y 392.779,Z 756.19,A -85,B 0,C 180,E1 18644.295,E2 18644.295} C_VEL
LIN {X 0,Y 392.261,Z 763.433,A -85,B 0,C 180,E1 18641.021,E2 18641.021} C_VEL
LIN {X 0,Y 392.064,Z 768.316,A -85,B 0,C 180,E1 18638.063,E2 18638.063} C_VEL
LIN {X 0,Y 392.007,Z 771.774,A -85,B 0,C 180,E1 18634.975,E2 18634.975} C_VEL
LIN {X 0,Y 392.008,Z 773.506,A -85,B 0,C 180,E1 18632.046,E2 18632.046} C_VEL
LIN {X 0,Y 392.015,Z 773.755,A -85,B 0,C 180,E1 18628.977,E2 18628.977} C_VEL
LIN {X 0,Y 392.007,Z 772.464,A -85,B 0,C 180,E1 18626.051,E2 18626.051} C_VEL
LIN {X 0,Y 392.042,Z 769.514,A -85,B 0,C 180,E1 18622.968,E2 18622.968} C_VEL
LIN {X 0,Y 392.183,Z 764.826,A -85,B 0,C 180,E1 18619.868,E2 18619.868} C_VEL
LIN {X 0,Y 392.576,Z 758.366,A -85,B 0,C 180,E1 18616.748,E2 18616.748} C_VEL
LIN {X 0,Y 393.324,Z 749.936,A -85,B 0,C 180,E1 18613.61,E2 18613.61} C_VEL
LIN {X 0,Y 394.474,Z 739.948,A -85,B 0,C 180,E1 18610.607,E2 18610.607} C_VEL
LIN {X 0,Y 396.04,Z 728.488,A -85,B 0,C 180,E1 18607.747,E2 18607.747} C_VEL
LIN {X 0,Y 398.139,Z 714.791,A -85,B 0,C 180,E1 18604.886,E2 18604.886} C_VEL
LIN {X 0,Y 400.609,Z 699.895,A -85,B 0,C 180,E1 18602.259,E2 18602.259} C_VEL
LIN {X 0,Y 403.54,Z 682.909,A -85,B 0,C 180,E1 18599.72,E2 18599.72} C_VEL
LIN {X 0,Y 406.697,Z 664.663,A -85,B 0,C 180,E1 18597.424,E2 18597.424} C_VEL
LIN {X 0,Y 409.867,Z 646.105,A -85,B 0,C 180,E1 18595.446,E2 18595.446} C_VEL
LIN {X 0,Y 413.159,Z 625.936,A -85,B 0,C 180,E1 18593.636,E2 18593.636} C_VEL
LIN {X 0,Y 416.758,Z 603.284,A -85,B 0,C 180,E1 18591.933,E2 18591.933} C_VEL
LIN {X 0,Y 420.131,Z 580.931,A -85,B 0,C 180,E1 18590.548,E2 18590.548} C_VEL
LIN {X 0,Y 423.425,Z 557.49,A -85,B 0,C 180,E1 18589.383,E2 18589.383} C_VEL
LIN {X 0,Y 426.577,Z 533.041,A -85,B 0,C 180,E1 18588.433,E2 18588.433} C_VEL
LIN {X 0,Y 429.323,Z 505.715,A -85,B 0,C 180,E1 18587.634,E2 18587.634} C_VEL
LIN {X 0,Y 430.904,Z 485.571,A -85,B 0,C 180,E1 18587.223,E2 18587.223} C_VEL
LIN {X 0,Y 433.072,Z 463.43,A -85,B 0,C 180,E1 18586.989,E2 18586.989} C_VEL
LIN {X 0,Y 435.303,Z 443.526,A -85,B 0,C 180,E1 18586.805,E2 18586.805} C_VEL
LIN {X 0,Y 443.712,Z 419.692,A -85,B 0,C 180,E1 18586.048,E2 18586.048} C_VEL
LIN {X 0,Y 451.028,Z 398.874,A -85,B 0,C 180,E1 18585.401,E2 18585.401} C_VEL
LIN {X 0,Y 461.132,Z 374.914,A -85,B 0,C 180,E1 18584.844,E2 18584.844} C_VEL
LIN {X 0,Y 475.993,Z 343.989,A -85,B 0,C 180,E1 18584.336,E2 18584.336} C_VEL
LIN {X 0,Y 478.624,Z 338.461,A -85,B 0,C 180,E1 18584.245,E2 18584.245} C_VEL
LIN {X 0,Y 469.034,Z 329.211,A -85,B 0,C 180,E1 18582.654,E2 18582.654} C_VEL
LIN {X 0,Y 459.637,Z 316.986,A -85,B 0,C 180,E1 18580.737,E2 18580.737} C_VEL
LIN {X 0,Y 452.938,Z 304.628,A -85,B 0,C 180,E1 18578.986,E2 18578.986} C_VEL
LIN {X 0,Y 444.232,Z 282.232,A -85,B 0,C 180,E1 18575.976,E2 18575.976} C_VEL
LIN {X 0,Y 438.693,Z 285.483,A -85,B 0,C 180,E1 18575.374,E2 18575.374} C_VEL
LIN {X 0,Y 432.366,Z 289.358,A -85,B 0,C 180,E1 18574.672,E2 18574.672} C_VEL
LIN {X 0,Y 427.581,Z 292.356,A -85,B 0,C 180,E1 18574.126,E2 18574.126} C_VEL
LIN {X 0,Y 422.018,Z 296.141,A -85,B 0,C 180,E1 18573.491,E2 18573.491} C_VEL
LIN {X 0,Y 419.913,Z 297.229,A -85,B 0,C 180,E1 18573.206,E2 18573.206} C_VEL
LIN {X 0,Y 416.513,Z 300.046,A -85,B 0,C 180,E1 18572.839,E2 18572.839} C_VEL
LIN {X 0,Y 413.708,Z 301.294,A -85,B 0,C 180,E1 18572.386,E2 18572.386} C_VEL
LIN {X 0,Y 411.879,Z 344.375,A -85,B 0,C 180,E1 18568.411,E2 18568.411} C_VEL
LIN {X 0,Y 409.508,Z 354.567,A -85,B 0,C 180,E1 18567.718,E2 18567.718} C_VEL
LIN {X 0,Y 409.043,Z 359.922,A -85,B 0,C 180,E1 18567.545,E2 18567.545} C_VEL
LIN {X 0,Y 404.321,Z 461.117,A -85,B 0,C 180,E1 18565.006,E2 18565.006} C_VEL
LIN {X 0,Y 403.127,Z 508.9,A -85,B 0,C 180,E1 18563.875,E2 18563.875} C_VEL
LIN {X 0,Y 403.049,Z 528.168,A -85,B 0,C 180,E1 18563.284,E2 18563.284} C_VEL
LIN {X 0,Y 402.662,Z 545.338,A -85,B 0,C 180,E1 18562.482,E2 18562.482} C_VEL
LIN {X 0,Y 402.048,Z 561.95,A -85,B 0,C 180,E1 18561.443,E2 18561.443} C_VEL
LIN {X 0,Y 401.207,Z 577.209,A -85,B 0,C 180,E1 18560.191,E2 18560.191} C_VEL
LIN {X 0,Y 400.177,Z 592.082,A -85,B 0,C 180,E1 18558.651,E2 18558.651} C_VEL
LIN {X 0,Y 399.143,Z 604.461,A -85,B 0,C 180,E1 18557.042,E2 18557.042} C_VEL
LIN {X 0,Y 398.01,Z 616.186,A -85,B 0,C 180,E1 18555.145,E2 18555.145} C_VEL
LIN {X 0,Y 396.967,Z 626.248,A -85,B 0,C 180,E1 18553.102,E2 18553.102} C_VEL
LIN {X 0,Y 396.095,Z 634.093,A -85,B 0,C 180,E1 18551.06,E2 18551.06} C_VEL
LIN {X 0,Y 395.304,Z 640.913,A -85,B 0,C 180,E1 18548.728,E2 18548.728} C_VEL
LIN {X 0,Y 394.71,Z 645.774,A -85,B 0,C 180,E1 18546.399,E2 18546.399} C_VEL
LIN {X 0,Y 394.287,Z 648.777,A -85,B 0,C 180,E1 18544.071,E2 18544.071} C_VEL
LIN {X 0,Y 394.007,Z 650.155,A -85,B 0,C 180,E1 18541.599,E2 18541.599} C_VEL
LIN {X 0,Y 393.863,Z 649.728,A -85,B 0,C 180,E1 18539.127,E2 18539.127} C_VEL
LIN {X 0,Y 393.834,Z 647.415,A -85,B 0,C 180,E1 18536.638,E2 18536.638} C_VEL
LIN {X 0,Y 393.96,Z 643.307,A -85,B 0,C 180,E1 18534.173,E2 18534.173} C_VEL
LIN {X 0,Y 394.253,Z 637.63,A -85,B 0,C 180,E1 18531.835,E2 18531.835} C_VEL
LIN {X 0,Y 394.73,Z 629.948,A -85,B 0,C 180,E1 18529.491,E2 18529.491} C_VEL
LIN {X 0,Y 395.38,Z 620.717,A -85,B 0,C 180,E1 18527.29,E2 18527.29} C_VEL
LIN {X 0,Y 396.203,Z 609.938,A -85,B 0,C 180,E1 18525.233,E2 18525.233} C_VEL
LIN {X 0,Y 397.156,Z 597.544,A -85,B 0,C 180,E1 18523.321,E2 18523.321} C_VEL
LIN {X 0,Y 398.2,Z 583.477,A -85,B 0,C 180,E1 18521.555,E2 18521.555} C_VEL
LIN {X 0,Y 399.218,Z 568.08,A -85,B 0,C 180,E1 18520.009,E2 18520.009} C_VEL
LIN {X 0,Y 400.177,Z 551.488,A -85,B 0,C 180,E1 18518.682,E2 18518.682} C_VEL
LIN {X 0,Y 400.914,Z 534.613,A -85,B 0,C 180,E1 18517.645,E2 18517.645} C_VEL
LIN {X 0,Y 401.499,Z 516.107,A -85,B 0,C 180,E1 18516.813,E2 18516.813} C_VEL
LIN {X 0,Y 401.777,Z 497.934,A -85,B 0,C 180,E1 18516.274,E2 18516.274} C_VEL
LIN {X 0,Y 404.086,Z 397.871,A -85,B 0,C 180,E1 18514.183,E2 18514.183} C_VEL
LIN {X 0,Y 404.789,Z 399.232,A -85,B 0,C 180,E1 18514.011,E2 18514.011} C_VEL
LIN {X 0,Y 406.192,Z 398.959,A -85,B 0,C 180,E1 18513.778,E2 18513.778} C_VEL
LIN {X 0,Y 408.414,Z 395.639,A -85,B 0,C 180,E1 18513.52,E2 18513.52} C_VEL
LIN {X 0,Y 411.873,Z 386.78,A -85,B 0,C 180,E1 18513.252,E2 18513.252} C_VEL
LIN {X 0,Y 415.782,Z 372.746,A -85,B 0,C 180,E1 18513.079,E2 18513.079} C_VEL
LIN {X 0,Y 418.701,Z 369.627,A -85,B 0,C 180,E1 18512.709,E2 18512.709} C_VEL
LIN {X 0,Y 421.916,Z 363.542,A -85,B 0,C 180,E1 18512.399,E2 18512.399} C_VEL
LIN {X 0,Y 425.843,Z 352.375,A -85,B 0,C 180,E1 18512.139,E2 18512.139} C_VEL
LIN {X 0,Y 427.398,Z 346.965,A -85,B 0,C 180,E1 18512.065,E2 18512.065} C_VEL
LIN {X 0,Y 431.864,Z 343.147,A -85,B 0,C 180,E1 18511.514,E2 18511.514} C_VEL
LIN {X 0,Y 434.006,Z 342.416,A -85,B 0,C 180,E1 18511.229,E2 18511.229} C_VEL
LIN {X 0,Y 426.541,Z 484.263,A -85,B 0,C 180,E1 18508.186,E2 18508.186} C_VEL
LIN {X 0,Y 425.151,Z 505.864,A -85,B 0,C 180,E1 18507.484,E2 18507.484} C_VEL
LIN {X 0,Y 423.278,Z 525.747,A -85,B 0,C 180,E1 18506.606,E2 18506.606} C_VEL
LIN {X 0,Y 420.916,Z 544.957,A -85,B 0,C 180,E1 18505.516,E2 18505.516} C_VEL
LIN {X 0,Y 418.083,Z 564.118,A -85,B 0,C 180,E1 18504.168,E2 18504.168} C_VEL
LIN {X 0,Y 414.909,Z 582.811,A -85,B 0,C 180,E1 18502.565,E2 18502.565} C_VEL
LIN {X 0,Y 411.653,Z 600.117,A -85,B 0,C 180,E1 18500.789,E2 18500.789} C_VEL
LIN {X 0,Y 408.523,Z 615.551,A -85,B 0,C 180,E1 18498.916,E2 18498.916} C_VEL
LIN {X 0,Y 406.51,Z 621.277,A -85,B 0,C 180,E1 18498.234,E2 18498.234} C_VEL
LIN {X 0,Y 398.231,Z 635.571,A -85,B 0,C 180,E1 18496.584,E2 18496.584} C_VEL
LIN {X 0,Y 396.207,Z 640.64,A -85,B 0,C 180,E1 18495.799,E2 18495.799} C_VEL
LIN {X 0,Y 392.993,Z 654.791,A -85,B 0,C 180,E1 18493.097,E2 18493.097} C_VEL
LIN {X 0,Y 390.402,Z 666.77,A -85,B 0,C 180,E1 18490.388,E2 18490.388} C_VEL
LIN {X 0,Y 388.203,Z 677.695,A -85,B 0,C 180,E1 18487.434,E2 18487.434} C_VEL
LIN {X 0,Y 386.492,Z 687.093,A -85,B 0,C 180,E1 18484.331,E2 18484.331} C_VEL
LIN {X 0,Y 385.342,Z 694.632,A -85,B 0,C 180,E1 18481.262,E2 18481.262} C_VEL
LIN {X 0,Y 384.63,Z 700.804,A -85,B 0,C 180,E1 18478.068,E2 18478.068} C_VEL
LIN {X 0,Y 384.259,Z 705.262,A -85,B 0,C 180,E1 18474.932,E2 18474.932} C_VEL
LIN {X 0,Y 384.103,Z 708.148,A -85,B 0,C 180,E1 18471.854,E2 18471.854} C_VEL
LIN {X 0,Y 384.045,Z 709.727,A -85,B 0,C 180,E1 18468.677,E2 18468.677} C_VEL
LIN {X 0,Y 384.049,Z 709.777,A -85,B 0,C 180,E1 18465.71,E2 18465.71} C_VEL
LIN {X 0,Y 384.081,Z 708.399,A -85,B 0,C 180,E1 18462.479,E2 18462.479} C_VEL
LIN {X 0,Y 384.214,Z 705.727,A -85,B 0,C 180,E1 18459.436,E2 18459.436} C_VEL
LIN {X 0,Y 384.547,Z 701.365,A -85,B 0,C 180,E1 18456.27,E2 18456.27} C_VEL
LIN {X 0,Y 385.232,Z 695.191,A -85,B 0,C 180,E1 18452.976,E2 18452.976} C_VEL
LIN {X 0,Y 386.339,Z 687.666,A -85,B 0,C 180,E1 18449.852,E2 18449.852} C_VEL
LIN {X 0,Y 387.97,Z 678.317,A -85,B 0,C 180,E1 18446.75,E2 18446.75} C_VEL
LIN {X 0,Y 389.954,Z 668.141,A -85,B 0,C 180,E1 18443.966,E2 18443.966} C_VEL
LIN {X 0,Y 392.483,Z 656.185,A -85,B 0,C 180,E1 18441.208,E2 18441.208} C_VEL
LIN {X 0,Y 395.427,Z 642.94,A -85,B 0,C 180,E1 18438.625,E2 18438.625} C_VEL
LIN {X 0,Y 398.639,Z 628.185,A -85,B 0,C 180,E1 18436.215,E2 18436.215} C_VEL
LIN {X 0,Y 402.02,Z 612.363,A -85,B 0,C 180,E1 18434.028,E2 18434.028} C_VEL
LIN {X 0,Y 405.461,Z 595.438,A -85,B 0,C 180,E1 18432.047,E2 18432.047} C_VEL
LIN {X 0,Y 408.727,Z 578.203,A -85,B 0,C 180,E1 18430.345,E2 18430.345} C_VEL
LIN {X 0,Y 411.739,Z 560.025,A -85,B 0,C 180,E1 18428.862,E2 18428.862} C_VEL
LIN {X 0,Y 414.445,Z 541.258,A -85,B 0,C 180,E1 18427.593,E2 18427.593} C_VEL
LIN {X 0,Y 416.803,Z 521.969,A -85,B 0,C 180,E1 18426.534,E2 18426.534} C_VEL
LIN {X 0,Y 418.751,Z 500.819,A -85,B 0,C 180,E1 18425.64,E2 18425.64} C_VEL
LIN {X 0,Y 420.053,Z 479.791,A -85,B 0,C 180,E1 18425.003,E2 18425.003} C_VEL
LIN {X 0,Y 428.426,Z 317.726,A -85,B 0,C 180,E1 18421.574,E2 18421.574} C_VEL
LIN {X 0,Y 431.058,Z 258.374,A -85,B 0,C 180,E1 18420.38,E2 18420.38} C_VEL
LIN {X 0,Y 425.17,Z 249.897,A -85,B 0,C 180,E1 18419.364,E2 18419.364} C_VEL
LIN {X 0,Y 412.191,Z 234.194,A -85,B 0,C 180,E1 18417.067,E2 18417.067} C_VEL
LIN {X 0,Y 402.378,Z 223.038,A -85,B 0,C 180,E1 18415.211,E2 18415.211} C_VEL
LIN {X 0,Y 400.871,Z 221.266,A -85,B 0,C 180,E1 18414.896,E2 18414.896} C_VEL
LIN {X 0,Y 398.831,Z 217.525,A -85,B 0,C 180,E1 18413.829,E2 18413.829} C_VEL
LIN {X 0,Y 396.887,Z 213.833,A -85,B 0,C 180,E1 18412.759,E2 18412.759} C_VEL
LIN {X 0,Y 394.012,Z 208.782,A -85,B 0,C 180,E1 18411.175,E2 18411.175} C_VEL
LIN {X 0,Y 391.321,Z 203.963,A -85,B 0,C 180,E1 18409.59,E2 18409.59} C_VEL
LIN {X 0,Y 389.097,Z 200.311,A -85,B 0,C 180,E1 18408.276,E2 18408.276} C_VEL
LIN {X 0,Y 388.411,Z 198.834,A -85,B 0,C 180,E1 18407.788,E2 18407.788} C_VEL
LIN {X 0,Y 386.142,Z 195.724,A -85,B 0,C 180,E1 18406.468,E2 18406.468} C_VEL
LIN {X 0,Y 385.615,Z 193.691,A -85,B 0,C 180,E1 18405.84,E2 18405.84} C_VEL
LIN {X 0,Y 385.616,Z 193.687,A -85,B 0,C 180,E1 18401.788,E2 18401.788} C_VEL
LIN {X 0,Y 385.597,Z 193.696,A -85,B 0,C 180,E1 18397.92,E2 18397.92} C_VEL
LIN {X 0,Y 385.568,Z 193.707,A -85,B 0,C 180,E1 18393.887,E2 18393.887} C_VEL
LIN {X 0,Y 385.585,Z 193.706,A -85,B 0,C 180,E1 18389.86,E2 18389.86} C_VEL
LIN {X 0,Y 385.611,Z 193.696,A -85,B 0,C 180,E1 18385.825,E2 18385.825} C_VEL
LIN {X 0,Y 385.625,Z 193.681,A -85,B 0,C 180,E1 18381.764,E2 18381.764} C_VEL
LIN {X 0,Y 385.599,Z 193.678,A -85,B 0,C 180,E1 18377.817,E2 18377.817} C_VEL
LIN {X 0,Y 385.572,Z 193.683,A -85,B 0,C 180,E1 18373.956,E2 18373.956} C_VEL
LIN {X 0,Y 385.581,Z 193.691,A -85,B 0,C 180,E1 18369.855,E2 18369.855} C_VEL
LIN {X 0,Y 385.605,Z 193.696,A -85,B 0,C 180,E1 18365.805,E2 18365.805} C_VEL
LIN {X 0,Y 385.623,Z 193.701,A -85,B 0,C 180,E1 18361.784,E2 18361.784} C_VEL
LIN {X 0,Y 385.608,Z 193.705,A -85,B 0,C 180,E1 18357.771,E2 18357.771} C_VEL
LIN {X 0,Y 385.573,Z 193.708,A -85,B 0,C 180,E1 18353.748,E2 18353.748} C_VEL
LIN {X 0,Y 385.585,Z 193.745,A -85,B 0,C 180,E1 18352.026,E2 18352.026} C_VEL
LIN {X 0,Y 386.662,Z 196.834,A -85,B 0,C 180,E1 18351.075,E2 18351.075} C_VEL
LIN {X 0,Y 388.793,Z 199.391,A -85,B 0,C 180,E1 18349.929,E2 18349.929} C_VEL
LIN {X 0,Y 390.485,Z 202.967,A -85,B 0,C 180,E1 18348.779,E2 18348.779} C_VEL
LIN {X 0,Y 391.859,Z 204.786,A -85,B 0,C 180,E1 18348.073,E2 18348.073} C_VEL
LIN {X 0,Y 394.051,Z 208.814,A -85,B 0,C 180,E1 18346.8,E2 18346.8} C_VEL
LIN {X 0,Y 397.669,Z 215.258,A -85,B 0,C 180,E1 18344.842,E2 18344.842} C_VEL
LIN {X 0,Y 402.797,Z 224.765,A -85,B 0,C 180,E1 18342.223,E2 18342.223} C_VEL
LIN {X 0,Y 409.066,Z 236.881,A -85,B 0,C 180,E1 18339.243,E2 18339.243} C_VEL
LIN {X 0,Y 415.8,Z 251.047,A -85,B 0,C 180,E1 18336.173,E2 18336.173} C_VEL
LIN {X 0,Y 423.146,Z 267.245,A -85,B 0,C 180,E1 18333.02,E2 18333.02} C_VEL
LIN {X 0,Y 427.528,Z 277.87,A -85,B 0,C 180,E1 18331.157,E2 18331.157} C_VEL
LIN {X 0,Y 421.737,Z 326.962,A -85,B 0,C 180,E1 18326.632,E2 18326.632} C_VEL
LIN {X 0,Y 421.612,Z 347.035,A -85,B 0,C 180,E1 18324.562,E2 18324.562} C_VEL
LIN {X 0,Y 423.49,Z 364.713,A -85,B 0,C 180,E1 18322.559,E2 18322.559} C_VEL
LIN {X 0,Y 427.411,Z 381.518,A -85,B 0,C 180,E1 18320.484,E2 18320.484} C_VEL
LIN {X 0,Y 433.082,Z 396.341,A -85,B 0,C 180,E1 18318.502,E2 18318.502} C_VEL
LIN {X 0,Y 440.574,Z 409.848,A -85,B 0,C 180,E1 18316.557,E2 18316.557} C_VEL
LIN {X 0,Y 448.296,Z 420.418,A -85,B 0,C 180,E1 18314.936,E2 18314.936} C_VEL
LIN {X 0,Y 441.853,Z 431.102,A -85,B 0,C 180,E1 18314.547,E2 18314.547} C_VEL
LIN {X 0,Y 432.224,Z 448.102,A -85,B 0,C 180,E1 18313.854,E2 18313.854} C_VEL
LIN {X 0,Y 429.567,Z 453.867,A -85,B 0,C 180,E1 18313.612,E2 18313.612} C_VEL
LIN {X 0,Y 425.653,Z 479.517,A -85,B 0,C 180,E1 18313.507,E2 18313.507} C_VEL
LIN {X 0,Y 423.806,Z 498.285,A -85,B 0,C 180,E1 18313.246,E2 18313.246} C_VEL
LIN {X 0,Y 421.608,Z 524.878,A -85,B 0,C 180,E1 18312.554,E2 18312.554} C_VEL
LIN {X 0,Y 418.583,Z 549.486,A -85,B 0,C 180,E1 18311.701,E2 18311.701} C_VEL
LIN {X 0,Y 415.225,Z 573.555,A -85,B 0,C 180,E1 18310.599,E2 18310.599} C_VEL
LIN {X 0,Y 411.66,Z 597.009,A -85,B 0,C 180,E1 18309.241,E2 18309.241} C_VEL
LIN {X 0,Y 408.083,Z 618.962,A -85,B 0,C 180,E1 18307.685,E2 18307.685} C_VEL
LIN {X 0,Y 404.578,Z 639.39,A -85,B 0,C 180,E1 18305.941,E2 18305.941} C_VEL
LIN {X 0,Y 401.048,Z 658.921,A -85,B 0,C 180,E1 18303.949,E2 18303.949} C_VEL
LIN {X 0,Y 397.63,Z 677.481,A -85,B 0,C 180,E1 18301.704,E2 18301.704} C_VEL
